LIN {X 0,Y 532.097,Z 327.827,A -85,B 0,C 180,E1 -4167.409,E2 -4167.409} C_VEL
LIN {X 0,Y 531.058,Z 327.962,A -85,B 0,C 180,E1 -4168.039,E2 -4168.039} C_VEL
LIN {X 0,Y 530.975,Z 327.968,A -85,B 0,C 180,E1 -4168.253,E2 -4168.253} C_VEL
LIN {X 0,Y 530.963,Z 327.965,A -85,B 0,C 180,E1 -4171.079,E2 -4171.079} C_VEL
LIN {X 0,Y 530.992,Z 327.968,A -85,B 0,C 180,E1 -4173.773,E2 -4173.773} C_VEL
LIN {X 0,Y 530.956,Z 327.969,A -85,B 0,C 180,E1 -4176.559,E2 -4176.559} C_VEL
LIN {X 0,Y 530.976,Z 327.967,A -85,B 0,C 180,E1 -4179.444,E2 -4179.444} C_VEL
LIN {X 0,Y 530.968,Z 327.967,A -85,B 0,C 180,E1 -4182.458,E2 -4182.458} C_VEL
LIN {X 0,Y 530.973,Z 327.971,A -85,B 0,C 180,E1 -4185.451,E2 -4185.451} C_VEL
LIN {X 0,Y 530.968,Z 327.966,A -85,B 0,C 180,E1 -4188.561,E2 -4188.561} C_VEL
LIN {X 0,Y 530.954,Z 327.976,A -85,B 0,C 180,E1 -4191.528,E2 -4191.528} C_VEL
LIN {X 0,Y 530.951,Z 327.968,A -85,B 0,C 180,E1 -4194.379,E2 -4194.379} C_VEL
LIN {X 0,Y 530.949,Z 327.974,A -85,B 0,C 180,E1 -4197.131,E2 -4197.131} C_VEL
LIN {X 0,Y 530.937,Z 327.974,A -85,B 0,C 180,E1 -4199.8,E2 -4199.8} C_VEL
LIN {X 0,Y 530.958,Z 327.969,A -85,B 0,C 180,E1 -4202.479,E2 -4202.479} C_VEL
LIN {X 0,Y 530.948,Z 327.975,A -85,B 0,C 180,E1 -4205.773,E2 -4205.773} C_VEL
LIN {X 0,Y 530.99,Z 328.027,A -85,B 0,C 180,E1 -4206.376,E2 -4206.376} C_VEL
LIN {X 0,Y 532.426,Z 335.68,A -85,B 0,C 180,E1 -4207.685,E2 -4207.685} C_VEL
LIN {X 0,Y 532.144,Z 349.705,A -85,B 0,C 180,E1 -4209.916,E2 -4209.916} C_VEL
LIN {X 0,Y 531.819,Z 362.546,A -85,B 0,C 180,E1 -4211.93,E2 -4211.93} C_VEL
LIN {X 0,Y 533.948,Z 373.777,A -85,B 0,C 180,E1 -4212.162,E2 -4212.162} C_VEL
LIN {X 0,Y 533.273,Z 498.769,A -85,B 0,C 180,E1 -4213.883,E2 -4213.883} C_VEL
LIN {X 0,Y 533.071,Z 512.331,A -85,B 0,C 180,E1 -4214.2,E2 -4214.2} C_VEL
LIN {X 0,Y 532.83,Z 526.788,A -85,B 0,C 180,E1 -4214.703,E2 -4214.703} C_VEL
LIN {X 0,Y 532.556,Z 539.12,A -85,B 0,C 180,E1 -4215.282,E2 -4215.282} C_VEL
LIN {X 0,Y 532.195,Z 550.61,A -85,B 0,C 180,E1 -4215.956,E2 -4215.956} C_VEL
LIN {X 0,Y 531.879,Z 561.401,A -85,B 0,C 180,E1 -4216.726,E2 -4216.726} C_VEL
LIN {X 0,Y 531.585,Z 571.53,A -85,B 0,C 180,E1 -4217.593,E2 -4217.593} C_VEL
LIN {X 0,Y 531.34,Z 581.016,A -85,B 0,C 180,E1 -4218.555,E2 -4218.555} C_VEL
LIN {X 0,Y 531.011,Z 591.907,A -85,B 0,C 180,E1 -4219.899,E2 -4219.899} C_VEL
LIN {X 0,Y 530.824,Z 599.5,A -85,B 0,C 180,E1 -4221.049,E2 -4221.049} C_VEL
LIN {X 0,Y 530.706,Z 604.896,A -85,B 0,C 180,E1 -4222.006,E2 -4222.006} C_VEL
LIN {X 0,Y 530.576,Z 610.311,A -85,B 0,C 180,E1 -4223.152,E2 -4223.152} C_VEL
LIN {X 0,Y 530.567,Z 614.741,A -85,B 0,C 180,E1 -4224.297,E2 -4224.297} C_VEL
LIN {X 0,Y 530.449,Z 618.285,A -85,B 0,C 180,E1 -4225.439,E2 -4225.439} C_VEL
LIN {X 0,Y 530.498,Z 620.206,A -85,B 0,C 180,E1 -4226.201,E2 -4226.201} C_VEL
LIN {X 0,Y 530.41,Z 622.929,A -85,B 0,C 180,E1 -4227.721,E2 -4227.721} C_VEL
LIN {X 0,Y 530.34,Z 624.236,A -85,B 0,C 180,E1 -4229.24,E2 -4229.24} C_VEL
LIN {X 0,Y 530.342,Z 624.496,A -85,B 0,C 180,E1 -4229.999,E2 -4229.999} C_VEL
LIN {X 0,Y 530.357,Z 623.834,A -85,B 0,C 180,E1 -4231.518,E2 -4231.518} C_VEL
LIN {X 0,Y 530.451,Z 621.843,A -85,B 0,C 180,E1 -4233.037,E2 -4233.037} C_VEL
LIN {X 0,Y 530.497,Z 620.436,A -85,B 0,C 180,E1 -4233.797,E2 -4233.797} C_VEL
LIN {X 0,Y 530.514,Z 616.296,A -85,B 0,C 180,E1 -4235.32,E2 -4235.32} C_VEL
LIN {X 0,Y 530.555,Z 613.779,A -85,B 0,C 180,E1 -4236.082,E2 -4236.082} C_VEL
LIN {X 0,Y 530.584,Z 609.106,A -85,B 0,C 180,E1 -4237.228,E2 -4237.228} C_VEL
LIN {X 0,Y 530.774,Z 602.297,A -85,B 0,C 180,E1 -4238.565,E2 -4238.565} C_VEL
LIN {X 0,Y 530.895,Z 595.198,A -85,B 0,C 180,E1 -4239.716,E2 -4239.716} C_VEL
LIN {X 0,Y 531.112,Z 588.237,A -85,B 0,C 180,E1 -4240.675,E2 -4240.675} C_VEL
LIN {X 0,Y 531.373,Z 579.159,A -85,B 0,C 180,E1 -4241.733,E2 -4241.733} C_VEL
LIN {X 0,Y 531.673,Z 569.372,A -85,B 0,C 180,E1 -4242.694,E2 -4242.694} C_VEL
LIN {X 0,Y 531.999,Z 557.577,A -85,B 0,C 180,E1 -4243.657,E2 -4243.657} C_VEL
LIN {X 0,Y 532.405,Z 544.281,A -85,B 0,C 180,E1 -4244.524,E2 -4244.524} C_VEL
LIN {X 0,Y 532.681,Z 532.145,A -85,B 0,C 180,E1 -4245.152,E2 -4245.152} C_VEL
LIN {X 0,Y 532.957,Z 519.572,A -85,B 0,C 180,E1 -4245.658,E2 -4245.658} C_VEL
LIN {X 0,Y 533.227,Z 505.576,A -85,B 0,C 180,E1 -4246.067,E2 -4246.067} C_VEL
LIN {X 0,Y 533.387,Z 488.986,A -85,B 0,C 180,E1 -4246.357,E2 -4246.357} C_VEL
LIN {X 0,Y 533.825,Z 373.018,A -85,B 0,C 180,E1 -4247.943,E2 -4247.943} C_VEL
LIN {X 0,Y 531.823,Z 362.504,A -85,B 0,C 180,E1 -4248.166,E2 -4248.166} C_VEL
LIN {X 0,Y 532.283,Z 343.943,A -85,B 0,C 180,E1 -4251.086,E2 -4251.086} C_VEL
LIN {X 0,Y 532.334,Z 335.057,A -85,B 0,C 180,E1 -4252.51,E2 -4252.51} C_VEL
LIN {X 0,Y 530.967,Z 327.972,A -85,B 0,C 180,E1 -4253.76,E2 -4253.76} C_VEL
LIN {X 0,Y 530.94,Z 327.977,A -85,B 0,C 180,E1 -4256.746,E2 -4256.746} C_VEL
LIN {X 0,Y 530.949,Z 327.974,A -85,B 0,C 180,E1 -4259.323,E2 -4259.323} C_VEL
LIN {X 0,Y 530.95,Z 327.97,A -85,B 0,C 180,E1 -4262.097,E2 -4262.097} C_VEL
LIN {X 0,Y 530.959,Z 327.976,A -85,B 0,C 180,E1 -4264.849,E2 -4264.849} C_VEL
LIN {X 0,Y 530.953,Z 327.969,A -85,B 0,C 180,E1 -4267.507,E2 -4267.507} C_VEL
LIN {X 0,Y 530.94,Z 327.972,A -85,B 0,C 180,E1 -4270.435,E2 -4270.435} C_VEL
LIN {X 0,Y 530.916,Z 327.973,A -85,B 0,C 180,E1 -4273.497,E2 -4273.497} C_VEL
LIN {X 0,Y 530.928,Z 327.974,A -85,B 0,C 180,E1 -4276.501,E2 -4276.501} C_VEL
LIN {X 0,Y 530.942,Z 327.97,A -85,B 0,C 180,E1 -4279.563,E2 -4279.563} C_VEL
LIN {X 0,Y 530.952,Z 327.97,A -85,B 0,C 180,E1 -4282.577,E2 -4282.577} C_VEL
LIN {X 0,Y 530.955,Z 327.968,A -85,B 0,C 180,E1 -4285.307,E2 -4285.307} C_VEL
LIN {X 0,Y 530.944,Z 327.965,A -85,B 0,C 180,E1 -4288.03,E2 -4288.03} C_VEL
LIN {X 0,Y 530.949,Z 327.974,A -85,B 0,C 180,E1 -4290.878,E2 -4290.878} C_VEL
LIN {X 0,Y 530.94,Z 327.965,A -85,B 0,C 180,E1 -4293.253,E2 -4293.253} C_VEL
LIN {X 0,Y 530.939,Z 327.969,A -85,B 0,C 180,E1 -4295.968,E2 -4295.968} C_VEL
LIN {X 0,Y 530.979,Z 327.964,A -85,B 0,C 180,E1 -4299.061,E2 -4299.061} C_VEL
LIN {X 0,Y 530.955,Z 327.963,A -85,B 0,C 180,E1 -4301.477,E2 -4301.477} C_VEL
LIN {X 0,Y 530.968,Z 327.974,A -85,B 0,C 180,E1 -4304.649,E2 -4304.649} C_VEL
LIN {X 0,Y 531,Z 327.961,A -85,B 0,C 180,E1 -4307.774,E2 -4307.774} C_VEL
LIN {X 0,Y 530.95,Z 327.969,A -85,B 0,C 180,E1 -4310.091,E2 -4310.091} C_VEL
LIN {X 0,Y 530.994,Z 327.967,A -85,B 0,C 180,E1 -4312.394,E2 -4312.394} C_VEL
LIN {X 0,Y 531.068,Z 327.959,A -85,B 0,C 180,E1 -4314.685,E2 -4314.685} C_VEL
LIN {X 0,Y 531.11,Z 327.948,A -85,B 0,C 180,E1 -4317.725,E2 -4317.725} C_VEL
LIN {X 0,Y 531.134,Z 327.951,A -85,B 0,C 180,E1 -4320.758,E2 -4320.758} C_VEL
LIN {X 0,Y 531.07,Z 327.954,A -85,B 0,C 180,E1 -4323.034,E2 -4323.034} C_VEL
LIN {X 0,Y 531.026,Z 327.961,A -85,B 0,C 180,E1 -4326.078,E2 -4326.078} C_VEL
LIN {X 0,Y 530.986,Z 327.964,A -85,B 0,C 180,E1 -4329.139,E2 -4329.139} C_VEL
LIN {X 0,Y 530.998,Z 327.967,A -85,B 0,C 180,E1 -4332.226,E2 -4332.226} C_VEL
LIN {X 0,Y 530.97,Z 327.965,A -85,B 0,C 180,E1 -4335.35,E2 -4335.35} C_VEL
LIN {X 0,Y 530.955,Z 327.975,A -85,B 0,C 180,E1 -4338.522,E2 -4338.522} C_VEL
LIN {X 0,Y 530.982,Z 327.962,A -85,B 0,C 180,E1 -4340.939,E2 -4340.939} C_VEL
LIN {X 0,Y 530.935,Z 327.973,A -85,B 0,C 180,E1 -4344.227,E2 -4344.227} C_VEL
LIN {X 0,Y 530.934,Z 327.972,A -85,B 0,C 180,E1 -4346.748,E2 -4346.748} C_VEL
LIN {X 0,Y 530.963,Z 327.962,A -85,B 0,C 180,E1 -4349.324,E2 -4349.324} C_VEL
LIN {X 0,Y 530.941,Z 327.974,A -85,B 0,C 180,E1 -4352.099,E2 -4352.099} C_VEL
LIN {X 0,Y 530.942,Z 327.971,A -85,B 0,C 180,E1 -4354.85,E2 -4354.85} C_VEL
LIN {X 0,Y 530.916,Z 327.973,A -85,B 0,C 180,E1 -4357.512,E2 -4357.512} C_VEL
LIN {X 0,Y 530.904,Z 327.98,A -85,B 0,C 180,E1 -4360.44,E2 -4360.44} C_VEL
LIN {X 0,Y 530.914,Z 327.973,A -85,B 0,C 180,E1 -4363.5,E2 -4363.5} C_VEL
LIN {X 0,Y 530.95,Z 327.97,A -85,B 0,C 180,E1 -4365.625,E2 -4365.625} C_VEL
LIN {X 0,Y 530.897,Z 327.98,A -85,B 0,C 180,E1 -4368.557,E2 -4368.557} C_VEL
LIN {X 0,Y 530.921,Z 327.973,A -85,B 0,C 180,E1 -4371.528,E2 -4371.528} C_VEL
LIN {X 0,Y 530.919,Z 327.979,A -85,B 0,C 180,E1 -4374.379,E2 -4374.379} C_VEL
LIN {X 0,Y 530.946,Z 327.969,A -85,B 0,C 180,E1 -4377.134,E2 -4377.134} C_VEL
LIN {X 0,Y 530.939,Z 327.974,A -85,B 0,C 180,E1 -4379.803,E2 -4379.803} C_VEL
LIN {X 0,Y 530.947,Z 327.974,A -85,B 0,C 180,E1 -4382.482,E2 -4382.482} C_VEL
LIN {X 0,Y 530.987,Z 328.019,A -85,B 0,C 180,E1 -4385.231,E2 -4385.231} C_VEL
LIN {X 0,Y 532.666,Z 336.952,A -85,B 0,C 180,E1 -4386.684,E2 -4386.684} C_VEL
LIN {X 0,Y 532.256,Z 355.336,A -85,B 0,C 180,E1 -4389.448,E2 -4389.448} C_VEL
LIN {X 0,Y 531.861,Z 371.775,A -85,B 0,C 180,E1 -4391.88,E2 -4391.88} C_VEL
LIN {X 0,Y 533.925,Z 383.626,A -85,B 0,C 180,E1 -4392.12,E2 -4392.12} C_VEL
LIN {X 0,Y 533.281,Z 508.566,A -85,B 0,C 180,E1 -4393.837,E2 -4393.837} C_VEL
LIN {X 0,Y 533.082,Z 523.14,A -85,B 0,C 180,E1 -4394.187,E2 -4394.187} C_VEL
LIN {X 0,Y 532.839,Z 536.02,A -85,B 0,C 180,E1 -4394.638,E2 -4394.638} C_VEL
LIN {X 0,Y 532.557,Z 548.002,A -85,B 0,C 180,E1 -4395.187,E2 -4395.187} C_VEL
LIN {X 0,Y 532.167,Z 561.163,A -85,B 0,C 180,E1 -4395.957,E2 -4395.957} C_VEL
LIN {X 0,Y 531.821,Z 573.057,A -85,B 0,C 180,E1 -4396.824,E2 -4396.824} C_VEL
LIN {X 0,Y 531.473,Z 583.923,A -85,B 0,C 180,E1 -4397.786,E2 -4397.786} C_VEL
LIN {X 0,Y 531.233,Z 594.661,A -85,B 0,C 180,E1 -4398.942,E2 -4398.942} C_VEL
LIN {X 0,Y 530.932,Z 603.524,A -85,B 0,C 180,E1 -4400.092,E2 -4400.092} C_VEL
LIN {X 0,Y 530.755,Z 612.018,A -85,B 0,C 180,E1 -4401.434,E2 -4401.434} C_VEL
LIN {X 0,Y 530.585,Z 618.859,A -85,B 0,C 180,E1 -4402.772,E2 -4402.772} C_VEL
LIN {X 0,Y 530.584,Z 624.963,A -85,B 0,C 180,E1 -4404.3,E2 -4404.3} C_VEL
LIN {X 0,Y 530.449,Z 628.45,A -85,B 0,C 180,E1 -4405.442,E2 -4405.442} C_VEL
LIN {X 0,Y 530.452,Z 631.838,A -85,B 0,C 180,E1 -4406.963,E2 -4406.963} C_VEL
LIN {X 0,Y 530.357,Z 633.838,A -85,B 0,C 180,E1 -4408.482,E2 -4408.482} C_VEL
LIN {X 0,Y 530.341,Z 634.5,A -85,B 0,C 180,E1 -4410.001,E2 -4410.001} C_VEL
LIN {X 0,Y 530.357,Z 633.834,A -85,B 0,C 180,E1 -4411.52,E2 -4411.52} C_VEL
LIN {X 0,Y 530.452,Z 631.83,A -85,B 0,C 180,E1 -4413.039,E2 -4413.039} C_VEL
LIN {X 0,Y 530.449,Z 628.44,A -85,B 0,C 180,E1 -4414.561,E2 -4414.561} C_VEL
LIN {X 0,Y 530.537,Z 623.565,A -85,B 0,C 180,E1 -4416.084,E2 -4416.084} C_VEL
LIN {X 0,Y 530.642,Z 617.036,A -85,B 0,C 180,E1 -4417.612,E2 -4417.612} C_VEL
LIN {X 0,Y 530.812,Z 609.768,A -85,B 0,C 180,E1 -4418.951,E2 -4418.951} C_VEL
LIN {X 0,Y 531.019,Z 600.768,A -85,B 0,C 180,E1 -4420.293,E2 -4420.293} C_VEL
LIN {X 0,Y 531.307,Z 591.32,A -85,B 0,C 180,E1 -4421.445,E2 -4421.445} C_VEL
LIN {X 0,Y 531.581,Z 580.861,A -85,B 0,C 180,E1 -4422.504,E2 -4422.504} C_VEL
LIN {X 0,Y 531.931,Z 569.317,A -85,B 0,C 180,E1 -4423.467,E2 -4423.467} C_VEL
LIN {X 0,Y 532.307,Z 556.508,A -85,B 0,C 180,E1 -4424.334,E2 -4424.334} C_VEL
LIN {X 0,Y 532.616,Z 544.007,A -85,B 0,C 180,E1 -4425.009,E2 -4425.009} C_VEL
LIN {X 0,Y 532.95,Z 530.331,A -85,B 0,C 180,E1 -4425.578,E2 -4425.578} C_VEL
LIN {X 0,Y 533.214,Z 516.18,A -85,B 0,C 180,E1 -4426.001,E2 -4426.001} C_VEL
LIN {X 0,Y 533.348,Z 502.389,A -85,B 0,C 180,E1 -4426.262,E2 -4426.262} C_VEL
LIN {X 0,Y 533.893,Z 383.182,A -85,B 0,C 180,E1 -4427.888,E2 -4427.888} C_VEL
LIN {X 0,Y 531.827,Z 371.698,A -85,B 0,C 180,E1 -4428.132,E2 -4428.132} C_VEL
LIN {X 0,Y 532.332,Z 351.756,A -85,B 0,C 180,E1 -4431.087,E2 -4431.087} C_VEL
LIN {X 0,Y 532.692,Z 336.936,A -85,B 0,C 180,E1 -4433.317,E2 -4433.317} C_VEL
LIN {X 0,Y 530.96,Z 327.973,A -85,B 0,C 180,E1 -4434.799,E2 -4434.799} C_VEL
LIN {X 0,Y 530.953,Z 327.976,A -85,B 0,C 180,E1 -4437.6,E2 -4437.6} C_VEL
LIN {X 0,Y 530.963,Z 327.968,A -85,B 0,C 180,E1 -4440.643,E2 -4440.643} C_VEL
LIN {X 0,Y 530.991,Z 327.967,A -85,B 0,C 180,E1 -4443.773,E2 -4443.773} C_VEL
LIN {X 0,Y 530.955,Z 327.969,A -85,B 0,C 180,E1 -4446.559,E2 -4446.559} C_VEL
LIN {X 0,Y 530.992,Z 327.967,A -85,B 0,C 180,E1 -4449.444,E2 -4449.444} C_VEL
LIN {X 0,Y 530.983,Z 327.967,A -85,B 0,C 180,E1 -4452.457,E2 -4452.457} C_VEL
LIN {X 0,Y 530.99,Z 327.964,A -85,B 0,C 180,E1 -4455.622,E2 -4455.622} C_VEL
LIN {X 0,Y 530.998,Z 327.969,A -85,B 0,C 180,E1 -4458.565,E2 -4458.565} C_VEL
LIN {X 0,Y 530.959,Z 327.967,A -85,B 0,C 180,E1 -4461.529,E2 -4461.529} C_VEL
LIN {X 0,Y 530.955,Z 327.976,A -85,B 0,C 180,E1 -4464.38,E2 -4464.38} C_VEL
LIN {X 0,Y 530.972,Z 327.967,A -85,B 0,C 180,E1 -4467.134,E2 -4467.134} C_VEL
LIN {X 0,Y 530.973,Z 327.971,A -85,B 0,C 180,E1 -4469.803,E2 -4469.803} C_VEL
LIN {X 0,Y 530.967,Z 327.973,A -85,B 0,C 180,E1 -4472.478,E2 -4472.478} C_VEL
LIN {X 0,Y 530.953,Z 327.97,A -85,B 0,C 180,E1 -4474.94,E2 -4474.94} C_VEL
LIN {X 0,Y 531.01,Z 328.064,A -85,B 0,C 180,E1 -4477.727,E2 -4477.727} C_VEL
LIN {X 0,Y 531.898,Z 334.003,A -85,B 0,C 180,E1 -4478.693,E2 -4478.693} C_VEL
LIN {X 0,Y 531.705,Z 352.894,A -85,B 0,C 180,E1 -4481.693,E2 -4481.693} C_VEL
LIN {X 0,Y 531.526,Z 365.213,A -85,B 0,C 180,E1 -4483.682,E2 -4483.682} C_VEL
LIN {X 0,Y 531.36,Z 373.68,A -85,B 0,C 180,E1 -4485.109,E2 -4485.109} C_VEL
LIN {X 0,Y 532.805,Z 383.09,A -85,B 0,C 180,E1 -4485.296,E2 -4485.296} C_VEL
LIN {X 0,Y 532.327,Z 480.991,A -85,B 0,C 180,E1 -4486.666,E2 -4486.666} C_VEL
LIN {X 0,Y 532.189,Z 494.465,A -85,B 0,C 180,E1 -4487.002,E2 -4487.002} C_VEL
LIN {X 0,Y 531.981,Z 506.626,A -85,B 0,C 180,E1 -4487.458,E2 -4487.458} C_VEL
LIN {X 0,Y 531.77,Z 518.851,A -85,B 0,C 180,E1 -4488.081,E2 -4488.081} C_VEL
LIN {X 0,Y 531.541,Z 530.473,A -85,B 0,C 180,E1 -4488.85,E2 -4488.85} C_VEL
LIN {X 0,Y 531.248,Z 540.771,A -85,B 0,C 180,E1 -4489.712,E2 -4489.712} C_VEL
LIN {X 0,Y 531.073,Z 550.146,A -85,B 0,C 180,E1 -4490.671,E2 -4490.671} C_VEL
LIN {X 0,Y 530.853,Z 557.738,A -85,B 0,C 180,E1 -4491.626,E2 -4491.626} C_VEL
LIN {X 0,Y 530.703,Z 565.237,A -85,B 0,C 180,E1 -4492.773,E2 -4492.773} C_VEL
LIN {X 0,Y 530.63,Z 571.198,A -85,B 0,C 180,E1 -4493.918,E2 -4493.918} C_VEL
LIN {X 0,Y 530.469,Z 575.952,A -85,B 0,C 180,E1 -4495.06,E2 -4495.06} C_VEL
LIN {X 0,Y 530.517,Z 579.514,A -85,B 0,C 180,E1 -4496.202,E2 -4496.202} C_VEL
LIN {X 0,Y 530.471,Z 581.366,A -85,B 0,C 180,E1 -4496.962,E2 -4496.962} C_VEL
LIN {X 0,Y 530.362,Z 583.823,A -85,B 0,C 180,E1 -4498.481,E2 -4498.481} C_VEL
LIN {X 0,Y 530.345,Z 584.454,A -85,B 0,C 180,E1 -4499.241,E2 -4499.241} C_VEL
LIN {X 0,Y 530.345,Z 584.674,A -85,B 0,C 180,E1 -4500,E2 -4500} C_VEL
LIN {X 0,Y 530.345,Z 584.483,A -85,B 0,C 180,E1 -4500.759,E2 -4500.759} C_VEL
LIN {X 0,Y 530.41,Z 582.917,A -85,B 0,C 180,E1 -4502.278,E2 -4502.278} C_VEL
LIN {X 0,Y 530.458,Z 581.543,A -85,B 0,C 180,E1 -4503.038,E2 -4503.038} C_VEL
LIN {X 0,Y 530.523,Z 578.711,A -85,B 0,C 180,E1 -4504.178,E2 -4504.178} C_VEL
LIN {X 0,Y 530.524,Z 574.814,A -85,B 0,C 180,E1 -4505.321,E2 -4505.321} C_VEL
LIN {X 0,Y 530.622,Z 568.966,A -85,B 0,C 180,E1 -4506.631,E2 -4506.631} C_VEL
LIN {X 0,Y 530.773,Z 562.224,A -85,B 0,C 180,E1 -4507.8,E2 -4507.8} C_VEL
LIN {X 0,Y 530.922,Z 554.043,A -85,B 0,C 180,E1 -4508.948,E2 -4508.948} C_VEL
LIN {X 0,Y 531.117,Z 545.592,A -85,B 0,C 180,E1 -4509.906,E2 -4509.906} C_VEL
LIN {X 0,Y 531.387,Z 535.209,A -85,B 0,C 180,E1 -4510.863,E2 -4510.863} C_VEL
LIN {X 0,Y 531.655,Z 524.494,A -85,B 0,C 180,E1 -4511.66,E2 -4511.66} C_VEL
LIN {X 0,Y 531.864,Z 513.565,A -85,B 0,C 180,E1 -4512.303,E2 -4512.303} C_VEL
LIN {X 0,Y 532.092,Z 500.687,A -85,B 0,C 180,E1 -4512.879,E2 -4512.879} C_VEL
LIN {X 0,Y 532.28,Z 487.641,A -85,B 0,C 180,E1 -4513.287,E2 -4513.287} C_VEL
LIN {X 0,Y 532.411,Z 473.759,A -85,B 0,C 180,E1 -4513.551,E2 -4513.551} C_VEL
LIN {X 0,Y 532.695,Z 381.43,A -85,B 0,C 180,E1 -4514.822,E2 -4514.822} C_VEL
LIN {X 0,Y 531.35,Z 373.456,A -85,B 0,C 180,E1 -4514.991,E2 -4514.991} C_VEL
LIN {X 0,Y 531.641,Z 356.128,A -85,B 0,C 180,E1 -4517.86,E2 -4517.86} C_VEL
LIN {X 0,Y 531.977,Z 337.651,A -85,B 0,C 180,E1 -4520.898,E2 -4520.898} C_VEL
LIN {X 0,Y 531.631,Z 331.341,A -85,B 0,C 180,E1 -4521.958,E2 -4521.958} C_VEL
LIN {X 0,Y 531,Z 327.97,A -85,B 0,C 180,E1 -4522.571,E2 -4522.571} C_VEL
LIN {X 0,Y 531.017,Z 327.965,A -85,B 0,C 180,E1 -4525.897,E2 -4525.897} C_VEL
LIN {X 0,Y 530.975,Z 327.968,A -85,B 0,C 180,E1 -4528.253,E2 -4528.253} C_VEL
LIN {X 0,Y 530.314,Z 328.054,A -85,B 0,C 180,E1 -4528.885,E2 -4528.885} C_VEL
LIN {X 0,Y 527.468,Z 328.408,A -85,B 0,C 180,E1 -4529.913,E2 -4529.913} C_VEL
LIN {X 0,Y 525.054,Z 328.706,A -85,B 0,C 180,E1 -4530.74,E2 -4530.74} C_VEL
LIN {X 0,Y 524.012,Z 328.833,A -85,B 0,C 180,E1 -4531.379,E2 -4531.379} C_VEL
LIN {X 0,Y 523.924,Z 328.844,A -85,B 0,C 180,E1 -4531.595,E2 -4531.595} C_VEL
LIN {X 0,Y 523.937,Z 328.847,A -85,B 0,C 180,E1 -4534.29,E2 -4534.29} C_VEL
LIN {X 0,Y 523.909,Z 328.845,A -85,B 0,C 180,E1 -4537.132,E2 -4537.132} C_VEL
LIN {X 0,Y 523.918,Z 328.849,A -85,B 0,C 180,E1 -4540.126,E2 -4540.126} C_VEL
LIN {X 0,Y 523.927,Z 328.844,A -85,B 0,C 180,E1 -4542.457,E2 -4542.457} C_VEL
LIN {X 0,Y 523.943,Z 328.845,A -85,B 0,C 180,E1 -4545.31,E2 -4545.31} C_VEL
LIN {X 0,Y 523.928,Z 328.843,A -85,B 0,C 180,E1 -4548.694,E2 -4548.694} C_VEL
LIN {X 0,Y 523.907,Z 328.85,A -85,B 0,C 180,E1 -4551.897,E2 -4551.897} C_VEL
LIN {X 0,Y 523.921,Z 328.846,A -85,B 0,C 180,E1 -4554.912,E2 -4554.912} C_VEL
LIN {X 0,Y 523.903,Z 328.852,A -85,B 0,C 180,E1 -4557.686,E2 -4557.686} C_VEL
LIN {X 0,Y 523.935,Z 328.845,A -85,B 0,C 180,E1 -4560.681,E2 -4560.681} C_VEL
LIN {X 0,Y 523.881,Z 328.854,A -85,B 0,C 180,E1 -4563.723,E2 -4563.723} C_VEL
LIN {X 0,Y 523.944,Z 328.855,A -85,B 0,C 180,E1 -4566.166,E2 -4566.166} C_VEL
LIN {X 0,Y 525.549,Z 337.744,A -85,B 0,C 180,E1 -4567.704,E2 -4567.704} C_VEL
LIN {X 0,Y 525.115,Z 353.578,A -85,B 0,C 180,E1 -4570.248,E2 -4570.248} C_VEL
LIN {X 0,Y 524.903,Z 362.629,A -85,B 0,C 180,E1 -4571.685,E2 -4571.685} C_VEL
LIN {X 0,Y 527.21,Z 375.245,A -85,B 0,C 180,E1 -4571.946,E2 -4571.946} C_VEL
LIN {X 0,Y 526.462,Z 500.288,A -85,B 0,C 180,E1 -4573.694,E2 -4573.694} C_VEL
LIN {X 0,Y 526.182,Z 514.907,A -85,B 0,C 180,E1 -4574.064,E2 -4574.064} C_VEL
LIN {X 0,Y 525.899,Z 529.12,A -85,B 0,C 180,E1 -4574.596,E2 -4574.596} C_VEL
LIN {X 0,Y 525.631,Z 540.988,A -85,B 0,C 180,E1 -4575.183,E2 -4575.183} C_VEL
LIN {X 0,Y 525.172,Z 553.604,A -85,B 0,C 180,E1 -4575.962,E2 -4575.962} C_VEL
LIN {X 0,Y 524.801,Z 566.277,A -85,B 0,C 180,E1 -4576.938,E2 -4576.938} C_VEL
LIN {X 0,Y 524.448,Z 576.751,A -85,B 0,C 180,E1 -4577.928,E2 -4577.928} C_VEL
LIN {X 0,Y 524.2,Z 586.052,A -85,B 0,C 180,E1 -4578.985,E2 -4578.985} C_VEL
LIN {X 0,Y 523.895,Z 594.661,A -85,B 0,C 180,E1 -4580.151,E2 -4580.151} C_VEL
LIN {X 0,Y 523.715,Z 601.848,A -85,B 0,C 180,E1 -4581.316,E2 -4581.316} C_VEL
LIN {X 0,Y 523.541,Z 608.743,A -85,B 0,C 180,E1 -4582.672,E2 -4582.672} C_VEL
LIN {X 0,Y 523.481,Z 614.831,A -85,B 0,C 180,E1 -4584.22,E2 -4584.22} C_VEL
LIN {X 0,Y 523.353,Z 618.372,A -85,B 0,C 180,E1 -4585.377,E2 -4585.377} C_VEL
LIN {X 0,Y 523.42,Z 620.275,A -85,B 0,C 180,E1 -4586.149,E2 -4586.149} C_VEL
LIN {X 0,Y 523.334,Z 622.991,A -85,B 0,C 180,E1 -4587.69,E2 -4587.69} C_VEL
LIN {X 0,Y 523.246,Z 624.3,A -85,B 0,C 180,E1 -4589.229,E2 -4589.229} C_VEL
LIN {X 0,Y 523.245,Z 624.544,A -85,B 0,C 180,E1 -4589.999,E2 -4589.999} C_VEL
LIN {X 0,Y 523.271,Z 623.893,A -85,B 0,C 180,E1 -4591.538,E2 -4591.538} C_VEL
LIN {X 0,Y 523.362,Z 621.913,A -85,B 0,C 180,E1 -4593.078,E2 -4593.078} C_VEL
LIN {X 0,Y 523.419,Z 620.489,A -85,B 0,C 180,E1 -4593.848,E2 -4593.848} C_VEL
LIN {X 0,Y 523.448,Z 616.381,A -85,B 0,C 180,E1 -4595.392,E2 -4595.392} C_VEL
LIN {X 0,Y 523.487,Z 612.36,A -85,B 0,C 180,E1 -4596.546,E2 -4596.546} C_VEL
LIN {X 0,Y 523.589,Z 607.34,A -85,B 0,C 180,E1 -4597.713,E2 -4597.713} C_VEL
LIN {X 0,Y 523.727,Z 601.259,A -85,B 0,C 180,E1 -4598.876,E2 -4598.876} C_VEL
LIN {X 0,Y 523.886,Z 593.962,A -85,B 0,C 180,E1 -4600.042,E2 -4600.042} C_VEL
LIN {X 0,Y 524.226,Z 585.231,A -85,B 0,C 180,E1 -4601.208,E2 -4601.208} C_VEL
LIN {X 0,Y 524.531,Z 574.611,A -85,B 0,C 180,E1 -4602.378,E2 -4602.378} C_VEL
LIN {X 0,Y 524.918,Z 562.676,A -85,B 0,C 180,E1 -4603.451,E2 -4603.451} C_VEL
LIN {X 0,Y 525.296,Z 550.638,A -85,B 0,C 180,E1 -4604.329,E2 -4604.329} C_VEL
LIN {X 0,Y 525.709,Z 537.267,A -85,B 0,C 180,E1 -4605.11,E2 -4605.11} C_VEL
LIN {X 0,Y 526.077,Z 523.353,A -85,B 0,C 180,E1 -4605.729,E2 -4605.729} C_VEL
LIN {X 0,Y 526.319,Z 509.807,A -85,B 0,C 180,E1 -4606.171,E2 -4606.171} C_VEL
LIN {X 0,Y 526.498,Z 495.634,A -85,B 0,C 180,E1 -4606.477,E2 -4606.477} C_VEL
LIN {X 0,Y 527.212,Z 374.976,A -85,B 0,C 180,E1 -4608.148,E2 -4608.148} C_VEL
LIN {X 0,Y 524.901,Z 362.492,A -85,B 0,C 180,E1 -4608.427,E2 -4608.427} C_VEL
LIN {X 0,Y 525.379,Z 343.995,A -85,B 0,C 180,E1 -4611.377,E2 -4611.377} C_VEL
LIN {X 0,Y 525.402,Z 336.262,A -85,B 0,C 180,E1 -4612.635,E2 -4612.635} C_VEL
LIN {X 0,Y 523.919,Z 328.85,A -85,B 0,C 180,E1 -4613.938,E2 -4613.938} C_VEL
LIN {X 0,Y 523.889,Z 328.856,A -85,B 0,C 180,E1 -4617.135,E2 -4617.135} C_VEL
LIN {X 0,Y 523.879,Z 328.852,A -85,B 0,C 180,E1 -4619.758,E2 -4619.758} C_VEL
LIN {X 0,Y 523.923,Z 328.848,A -85,B 0,C 180,E1 -4622.448,E2 -4622.448} C_VEL
LIN {X 0,Y 523.91,Z 328.851,A -85,B 0,C 180,E1 -4625.226,E2 -4625.226} C_VEL
LIN {X 0,Y 523.902,Z 328.846,A -85,B 0,C 180,E1 -4628.101,E2 -4628.101} C_VEL
LIN {X 0,Y 523.907,Z 328.849,A -85,B 0,C 180,E1 -4631.304,E2 -4631.304} C_VEL
LIN {X 0,Y 523.924,Z 328.849,A -85,B 0,C 180,E1 -4634.688,E2 -4634.688} C_VEL
LIN {X 0,Y 523.897,Z 328.846,A -85,B 0,C 180,E1 -4637.875,E2 -4637.875} C_VEL
LIN {X 0,Y 523.901,Z 328.848,A -85,B 0,C 180,E1 -4641.08,E2 -4641.08} C_VEL
LIN {X 0,Y 523.881,Z 328.848,A -85,B 0,C 180,E1 -4643.824,E2 -4643.824} C_VEL
LIN {X 0,Y 523.899,Z 328.852,A -85,B 0,C 180,E1 -4646.632,E2 -4646.632} C_VEL
LIN {X 0,Y 523.924,Z 328.844,A -85,B 0,C 180,E1 -4649.353,E2 -4649.353} C_VEL
LIN {X 0,Y 523.904,Z 328.847,A -85,B 0,C 180,E1 -4652.293,E2 -4652.293} C_VEL
LIN {X 0,Y 523.89,Z 328.847,A -85,B 0,C 180,E1 -4655.426,E2 -4655.426} C_VEL
LIN {X 0,Y 523.922,Z 328.843,A -85,B 0,C 180,E1 -4657.939,E2 -4657.939} C_VEL
LIN {X 0,Y 523.947,Z 328.841,A -85,B 0,C 180,E1 -4660.407,E2 -4660.407} C_VEL
LIN {X 0,Y 523.923,Z 328.849,A -85,B 0,C 180,E1 -4662.836,E2 -4662.836} C_VEL
LIN {X 0,Y 523.945,Z 328.842,A -85,B 0,C 180,E1 -4665.235,E2 -4665.235} C_VEL
LIN {X 0,Y 523.998,Z 328.838,A -85,B 0,C 180,E1 -4668.394,E2 -4668.394} C_VEL
LIN {X 0,Y 523.965,Z 328.836,A -85,B 0,C 180,E1 -4671.515,E2 -4671.515} C_VEL
LIN {X 0,Y 524.014,Z 328.838,A -85,B 0,C 180,E1 -4674.613,E2 -4674.613} C_VEL
LIN {X 0,Y 524.083,Z 328.823,A -85,B 0,C 180,E1 -4677.694,E2 -4677.694} C_VEL
LIN {X 0,Y 524.104,Z 328.826,A -85,B 0,C 180,E1 -4680.768,E2 -4680.768} C_VEL
LIN {X 0,Y 524.01,Z 328.833,A -85,B 0,C 180,E1 -4683.075,E2 -4683.075} C_VEL
LIN {X 0,Y 523.988,Z 328.838,A -85,B 0,C 180,E1 -4686.16,E2 -4686.16} C_VEL
LIN {X 0,Y 523.935,Z 328.841,A -85,B 0,C 180,E1 -4689.263,E2 -4689.263} C_VEL
LIN {X 0,Y 523.937,Z 328.849,A -85,B 0,C 180,E1 -4692.393,E2 -4692.393} C_VEL
LIN {X 0,Y 523.908,Z 328.845,A -85,B 0,C 180,E1 -4695.563,E2 -4695.563} C_VEL
LIN {X 0,Y 523.9,Z 328.847,A -85,B 0,C 180,E1 -4697.971,E2 -4697.971} C_VEL
LIN {X 0,Y 523.957,Z 328.844,A -85,B 0,C 180,E1 -4700.411,E2 -4700.411} C_VEL
LIN {X 0,Y 523.892,Z 328.846,A -85,B 0,C 180,E1 -4702.894,E2 -4702.894} C_VEL
LIN {X 0,Y 523.881,Z 328.848,A -85,B 0,C 180,E1 -4705.422,E2 -4705.422} C_VEL
LIN {X 0,Y 523.897,Z 328.849,A -85,B 0,C 180,E1 -4708.003,E2 -4708.003} C_VEL
LIN {X 0,Y 523.901,Z 328.85,A -85,B 0,C 180,E1 -4710.648,E2 -4710.648} C_VEL
LIN {X 0,Y 523.912,Z 328.845,A -85,B 0,C 180,E1 -4713.73,E2 -4713.73} C_VEL
LIN {X 0,Y 523.847,Z 328.861,A -85,B 0,C 180,E1 -4716.396,E2 -4716.396} C_VEL
LIN {X 0,Y 523.891,Z 328.848,A -85,B 0,C 180,E1 -4719.087,E2 -4719.087} C_VEL
LIN {X 0,Y 523.864,Z 328.857,A -85,B 0,C 180,E1 -4722.453,E2 -4722.453} C_VEL
LIN {X 0,Y 523.919,Z 328.844,A -85,B 0,C 180,E1 -4725.313,E2 -4725.313} C_VEL
LIN {X 0,Y 523.866,Z 328.854,A -85,B 0,C 180,E1 -4728.701,E2 -4728.701} C_VEL
LIN {X 0,Y 523.879,Z 328.854,A -85,B 0,C 180,E1 -4731.897,E2 -4731.897} C_VEL
LIN {X 0,Y 523.904,Z 328.847,A -85,B 0,C 180,E1 -4734.914,E2 -4734.914} C_VEL
LIN {X 0,Y 523.893,Z 328.851,A -85,B 0,C 180,E1 -4737.687,E2 -4737.687} C_VEL
LIN {X 0,Y 523.928,Z 328.844,A -85,B 0,C 180,E1 -4740.682,E2 -4740.682} C_VEL
LIN {X 0,Y 523.876,Z 328.855,A -85,B 0,C 180,E1 -4743.725,E2 -4743.725} C_VEL
LIN {X 0,Y 523.93,Z 328.968,A -85,B 0,C 180,E1 -4745.033,E2 -4745.033} C_VEL
LIN {X 0,Y 525.768,Z 338.244,A -85,B 0,C 180,E1 -4746.569,E2 -4746.569} C_VEL
LIN {X 0,Y 525.335,Z 355.89,A -85,B 0,C 180,E1 -4749.259,E2 -4749.259} C_VEL
LIN {X 0,Y 524.918,Z 371.725,A -85,B 0,C 180,E1 -4751.635,E2 -4751.635} C_VEL
LIN {X 0,Y 527.174,Z 384.814,A -85,B 0,C 180,E1 -4751.9,E2 -4751.9} C_VEL
LIN {X 0,Y 526.459,Z 509.734,A -85,B 0,C 180,E1 -4753.646,E2 -4753.646} C_VEL
LIN {X 0,Y 526.25,Z 523.912,A -85,B 0,C 180,E1 -4754.003,E2 -4754.003} C_VEL
LIN {X 0,Y 525.962,Z 536.173,A -85,B 0,C 180,E1 -4754.442,E2 -4754.442} C_VEL
LIN {X 0,Y 525.624,Z 549.71,A -85,B 0,C 180,E1 -4755.086,E2 -4755.086} C_VEL
LIN {X 0,Y 525.21,Z 562.523,A -85,B 0,C 180,E1 -4755.866,E2 -4755.866} C_VEL
LIN {X 0,Y 524.828,Z 574.164,A -85,B 0,C 180,E1 -4756.744,E2 -4756.744} C_VEL
LIN {X 0,Y 524.444,Z 585.359,A -85,B 0,C 180,E1 -4757.771,E2 -4757.771} C_VEL
LIN {X 0,Y 524.239,Z 594.593,A -85,B 0,C 180,E1 -4758.792,E2 -4758.792} C_VEL
LIN {X 0,Y 523.887,Z 603.456,A -85,B 0,C 180,E1 -4759.958,E2 -4759.958} C_VEL
LIN {X 0,Y 523.679,Z 611.95,A -85,B 0,C 180,E1 -4761.318,E2 -4761.318} C_VEL
LIN {X 0,Y 523.503,Z 618.791,A -85,B 0,C 180,E1 -4762.674,E2 -4762.674} C_VEL
LIN {X 0,Y 523.472,Z 623.507,A -85,B 0,C 180,E1 -4763.835,E2 -4763.835} C_VEL
LIN {X 0,Y 523.376,Z 627.329,A -85,B 0,C 180,E1 -4764.994,E2 -4764.994} C_VEL
LIN {X 0,Y 523.418,Z 630.275,A -85,B 0,C 180,E1 -4766.152,E2 -4766.152} C_VEL
LIN {X 0,Y 523.333,Z 632.966,A -85,B 0,C 180,E1 -4767.692,E2 -4767.692} C_VEL
LIN {X 0,Y 523.247,Z 634.296,A -85,B 0,C 180,E1 -4769.232,E2 -4769.232} C_VEL
LIN {X 0,Y 523.247,Z 634.295,A -85,B 0,C 180,E1 -4770.771,E2 -4770.771} C_VEL
LIN {X 0,Y 523.333,Z 632.959,A -85,B 0,C 180,E1 -4772.31,E2 -4772.31} C_VEL
LIN {X 0,Y 523.419,Z 630.265,A -85,B 0,C 180,E1 -4773.851,E2 -4773.851} C_VEL
LIN {X 0,Y 523.451,Z 626.139,A -85,B 0,C 180,E1 -4775.394,E2 -4775.394} C_VEL
LIN {X 0,Y 523.496,Z 620.451,A -85,B 0,C 180,E1 -4776.941,E2 -4776.941} C_VEL
LIN {X 0,Y 523.636,Z 614.034,A -85,B 0,C 180,E1 -4778.297,E2 -4778.297} C_VEL
LIN {X 0,Y 523.863,Z 606.064,A -85,B 0,C 180,E1 -4779.655,E2 -4779.655} C_VEL
LIN {X 0,Y 524.107,Z 597.725,A -85,B 0,C 180,E1 -4780.822,E2 -4780.822} C_VEL
LIN {X 0,Y 524.45,Z 586.943,A -85,B 0,C 180,E1 -4782.069,E2 -4782.069} C_VEL
LIN {X 0,Y 524.753,Z 576.485,A -85,B 0,C 180,E1 -4783.063,E2 -4783.063} C_VEL
LIN {X 0,Y 525.195,Z 563.913,A -85,B 0,C 180,E1 -4784.038,E2 -4784.038} C_VEL
LIN {X 0,Y 525.579,Z 551.436,A -85,B 0,C 180,E1 -4784.818,E2 -4784.818} C_VEL
LIN {X 0,Y 525.933,Z 538.617,A -85,B 0,C 180,E1 -4785.453,E2 -4785.453} C_VEL
LIN {X 0,Y 526.186,Z 524.835,A -85,B 0,C 180,E1 -4785.969,E2 -4785.969} C_VEL
LIN {X 0,Y 526.476,Z 510.769,A -85,B 0,C 180,E1 -4786.331,E2 -4786.331} C_VEL
LIN {X 0,Y 526.66,Z 482.647,A -85,B 0,C 180,E1 -4786.749,E2 -4786.749} C_VEL
LIN {X 0,Y 527.074,Z 383.404,A -85,B 0,C 180,E1 -4788.123,E2 -4788.123} C_VEL
LIN {X 0,Y 524.88,Z 371.609,A -85,B 0,C 180,E1 -4788.384,E2 -4788.384} C_VEL
LIN {X 0,Y 525.439,Z 351.694,A -85,B 0,C 180,E1 -4791.377,E2 -4791.377} C_VEL
LIN {X 0,Y 525.774,Z 338.227,A -85,B 0,C 180,E1 -4793.433,E2 -4793.433} C_VEL
LIN {X 0,Y 523.915,Z 328.851,A -85,B 0,C 180,E1 -4794.997,E2 -4794.997} C_VEL
LIN {X 0,Y 523.899,Z 328.852,A -85,B 0,C 180,E1 -4798.004,E2 -4798.004} C_VEL
LIN {X 0,Y 523.938,Z 328.845,A -85,B 0,C 180,E1 -4800.853,E2 -4800.853} C_VEL
LIN {X 0,Y 523.963,Z 328.843,A -85,B 0,C 180,E1 -4803.735,E2 -4803.735} C_VEL
LIN {X 0,Y 523.903,Z 328.847,A -85,B 0,C 180,E1 -4806.401,E2 -4806.401} C_VEL
LIN {X 0,Y 523.926,Z 328.85,A -85,B 0,C 180,E1 -4809.085,E2 -4809.085} C_VEL
LIN {X 0,Y 523.956,Z 328.84,A -85,B 0,C 180,E1 -4812.119,E2 -4812.119} C_VEL
LIN {X 0,Y 523.958,Z 328.842,A -85,B 0,C 180,E1 -4815.309,E2 -4815.309} C_VEL
LIN {X 0,Y 523.961,Z 328.846,A -85,B 0,C 180,E1 -4818.69,E2 -4818.69} C_VEL
LIN {X 0,Y 523.92,Z 328.846,A -85,B 0,C 180,E1 -4821.081,E2 -4821.081} C_VEL
LIN {X 0,Y 523.9,Z 328.848,A -85,B 0,C 180,E1 -4823.825,E2 -4823.825} C_VEL
LIN {X 0,Y 523.946,Z 328.846,A -85,B 0,C 180,E1 -4826.636,E2 -4826.636} C_VEL
LIN {X 0,Y 523.96,Z 328.842,A -85,B 0,C 180,E1 -4829.356,E2 -4829.356} C_VEL
LIN {X 0,Y 523.943,Z 328.85,A -85,B 0,C 180,E1 -4832.29,E2 -4832.29} C_VEL
LIN {X 0,Y 523.906,Z 328.851,A -85,B 0,C 180,E1 -4835.427,E2 -4835.427} C_VEL
LIN {X 0,Y 523.969,Z 328.926,A -85,B 0,C 180,E1 -4837.602,E2 -4837.602} C_VEL
LIN {X 0,Y 524.939,Z 335.046,A -85,B 0,C 180,E1 -4838.603,E2 -4838.603} C_VEL
LIN {X 0,Y 524.726,Z 353.072,A -85,B 0,C 180,E1 -4841.472,E2 -4841.472} C_VEL
LIN {X 0,Y 524.545,Z 366.585,A -85,B 0,C 180,E1 -4843.658,E2 -4843.658} C_VEL
LIN {X 0,Y 524.414,Z 374.134,A -85,B 0,C 180,E1 -4844.917,E2 -4844.917} C_VEL
LIN {X 0,Y 525.938,Z 383.216,A -85,B 0,C 180,E1 -4845.1,E2 -4845.1} C_VEL
LIN {X 0,Y 525.387,Z 482.607,A -85,B 0,C 180,E1 -4846.536,E2 -4846.536} C_VEL
LIN {X 0,Y 525.241,Z 494.834,A -85,B 0,C 180,E1 -4846.852,E2 -4846.852} C_VEL
LIN {X 0,Y 525.026,Z 507.5,A -85,B 0,C 180,E1 -4847.338,E2 -4847.338} C_VEL
LIN {X 0,Y 524.784,Z 519.803,A -85,B 0,C 180,E1 -4847.98,E2 -4847.98} C_VEL
LIN {X 0,Y 524.541,Z 531.774,A -85,B 0,C 180,E1 -4848.798,E2 -4848.798} C_VEL
LIN {X 0,Y 524.22,Z 541.925,A -85,B 0,C 180,E1 -4849.67,E2 -4849.67} C_VEL
LIN {X 0,Y 524.048,Z 550.305,A -85,B 0,C 180,E1 -4850.544,E2 -4850.544} C_VEL
LIN {X 0,Y 523.829,Z 557.958,A -85,B 0,C 180,E1 -4851.513,E2 -4851.513} C_VEL
LIN {X 0,Y 523.653,Z 565.482,A -85,B 0,C 180,E1 -4852.675,E2 -4852.675} C_VEL
LIN {X 0,Y 523.564,Z 571.478,A -85,B 0,C 180,E1 -4853.835,E2 -4853.835} C_VEL
LIN {X 0,Y 523.393,Z 576.24,A -85,B 0,C 180,E1 -4854.993,E2 -4854.993} C_VEL
LIN {X 0,Y 523.444,Z 579.827,A -85,B 0,C 180,E1 -4856.151,E2 -4856.151} C_VEL
LIN {X 0,Y 523.41,Z 581.692,A -85,B 0,C 180,E1 -4856.921,E2 -4856.921} C_VEL
LIN {X 0,Y 523.335,Z 583.121,A -85,B 0,C 180,E1 -4857.691,E2 -4857.691} C_VEL
LIN {X 0,Y 523.275,Z 584.15,A -85,B 0,C 180,E1 -4858.461,E2 -4858.461} C_VEL
LIN {X 0,Y 523.253,Z 584.776,A -85,B 0,C 180,E1 -4859.23,E2 -4859.23} C_VEL
LIN {X 0,Y 523.253,Z 584.997,A -85,B 0,C 180,E1 -4860,E2 -4860} C_VEL
LIN {X 0,Y 523.253,Z 584.812,A -85,B 0,C 180,E1 -4860.77,E2 -4860.77} C_VEL
LIN {X 0,Y 523.275,Z 584.223,A -85,B 0,C 180,E1 -4861.539,E2 -4861.539} C_VEL
LIN {X 0,Y 523.398,Z 581.849,A -85,B 0,C 180,E1 -4863.079,E2 -4863.079} C_VEL
LIN {X 0,Y 523.443,Z 578.996,A -85,B 0,C 180,E1 -4864.235,E2 -4864.235} C_VEL
LIN {X 0,Y 523.463,Z 575.076,A -85,B 0,C 180,E1 -4865.393,E2 -4865.393} C_VEL
LIN {X 0,Y 523.571,Z 569.657,A -85,B 0,C 180,E1 -4866.628,E2 -4866.628} C_VEL
LIN {X 0,Y 523.725,Z 562.425,A -85,B 0,C 180,E1 -4867.906,E2 -4867.906} C_VEL
LIN {X 0,Y 523.901,Z 554.19,A -85,B 0,C 180,E1 -4869.069,E2 -4869.069} C_VEL
LIN {X 0,Y 524.105,Z 545.718,A -85,B 0,C 180,E1 -4870.039,E2 -4870.039} C_VEL
LIN {X 0,Y 524.409,Z 535.27,A -85,B 0,C 180,E1 -4871.01,E2 -4871.01} C_VEL
LIN {X 0,Y 524.686,Z 524.931,A -85,B 0,C 180,E1 -4871.787,E2 -4871.787} C_VEL
LIN {X 0,Y 524.907,Z 513.442,A -85,B 0,C 180,E1 -4872.468,E2 -4872.468} C_VEL
LIN {X 0,Y 525.133,Z 501.708,A -85,B 0,C 180,E1 -4873.003,E2 -4873.003} C_VEL
LIN {X 0,Y 525.325,Z 489.075,A -85,B 0,C 180,E1 -4873.417,E2 -4873.417} C_VEL
LIN {X 0,Y 525.481,Z 476.067,A -85,B 0,C 180,E1 -4873.684,E2 -4873.684} C_VEL
LIN {X 0,Y 525.836,Z 382.364,A -85,B 0,C 180,E1 -4875.006,E2 -4875.006} C_VEL
LIN {X 0,Y 524.366,Z 373.657,A -85,B 0,C 180,E1 -4875.201,E2 -4875.201} C_VEL
LIN {X 0,Y 524.68,Z 356.766,A -85,B 0,C 180,E1 -4878.003,E2 -4878.003} C_VEL
LIN {X 0,Y 525.005,Z 338.886,A -85,B 0,C 180,E1 -4880.963,E2 -4880.963} C_VEL
LIN {X 0,Y 524.67,Z 332.584,A -85,B 0,C 180,E1 -4882.028,E2 -4882.028} C_VEL
LIN {X 0,Y 523.957,Z 328.847,A -85,B 0,C 180,E1 -4882.69,E2 -4882.69} C_VEL
LIN {X 0,Y 523.988,Z 328.842,A -85,B 0,C 180,E1 -4886.019,E2 -4886.019} C_VEL
LIN {X 0,Y 523.934,Z 328.843,A -85,B 0,C 180,E1 -4888.875,E2 -4888.875} C_VEL
LIN {X 0,Y 523.924,Z 328.844,A -85,B 0,C 180,E1 -4891.595,E2 -4891.595} C_VEL
LIN {X 0,Y 523.253,Z 328.933,A -85,B 0,C 180,E1 -4892.237,E2 -4892.237} C_VEL
LIN {X 0,Y 520.413,Z 329.282,A -85,B 0,C 180,E1 -4893.279,E2 -4893.279} C_VEL
LIN {X 0,Y 518.01,Z 329.588,A -85,B 0,C 180,E1 -4894.118,E2 -4894.118} C_VEL
LIN {X 0,Y 516.967,Z 329.711,A -85,B 0,C 180,E1 -4894.766,E2 -4894.766} C_VEL
LIN {X 0,Y 516.877,Z 329.721,A -85,B 0,C 180,E1 -4894.986,E2 -4894.986} C_VEL
LIN {X 0,Y 516.883,Z 329.728,A -85,B 0,C 180,E1 -4897.942,E2 -4897.942} C_VEL
LIN {X 0,Y 516.869,Z 329.722,A -85,B 0,C 180,E1 -4900.743,E2 -4900.743} C_VEL
LIN {X 0,Y 516.864,Z 329.723,A -85,B 0,C 180,E1 -4902.834,E2 -4902.834} C_VEL
LIN {X 0,Y 516.901,Z 329.719,A -85,B 0,C 180,E1 -4905.007,E2 -4905.007} C_VEL
LIN {X 0,Y 516.892,Z 329.72,A -85,B 0,C 180,E1 -4908.402,E2 -4908.402} C_VEL
LIN {X 0,Y 516.878,Z 329.727,A -85,B 0,C 180,E1 -4911.283,E2 -4911.283} C_VEL
LIN {X 0,Y 516.863,Z 329.724,A -85,B 0,C 180,E1 -4914.671,E2 -4914.671} C_VEL
LIN {X 0,Y 516.868,Z 329.729,A -85,B 0,C 180,E1 -4917.462,E2 -4917.462} C_VEL
LIN {X 0,Y 516.902,Z 329.722,A -85,B 0,C 180,E1 -4920.693,E2 -4920.693} C_VEL
LIN {X 0,Y 516.858,Z 329.729,A -85,B 0,C 180,E1 -4923.824,E2 -4923.824} C_VEL
LIN {X 0,Y 516.901,Z 329.867,A -85,B 0,C 180,E1 -4925.98,E2 -4925.98} C_VEL
LIN {X 0,Y 518.475,Z 337.7,A -85,B 0,C 180,E1 -4927.365,E2 -4927.365} C_VEL
LIN {X 0,Y 518.496,Z 346.027,A -85,B 0,C 180,E1 -4928.74,E2 -4928.74} C_VEL
LIN {X 0,Y 517.955,Z 362.666,A -85,B 0,C 180,E1 -4931.425,E2 -4931.425} C_VEL
LIN {X 0,Y 520.442,Z 376.303,A -85,B 0,C 180,E1 -4931.716,E2 -4931.716} C_VEL
LIN {X 0,Y 519.665,Z 499.169,A -85,B 0,C 180,E1 -4933.449,E2 -4933.449} C_VEL
LIN {X 0,Y 519.417,Z 513.612,A -85,B 0,C 180,E1 -4933.806,E2 -4933.806} C_VEL
LIN {X 0,Y 519.165,Z 526.942,A -85,B 0,C 180,E1 -4934.291,E2 -4934.291} C_VEL
LIN {X 0,Y 518.809,Z 539.323,A -85,B 0,C 180,E1 -4934.883,E2 -4934.883} C_VEL
LIN {X 0,Y 518.35,Z 552.262,A -85,B 0,C 180,E1 -4935.673,E2 -4935.673} C_VEL
LIN {X 0,Y 517.963,Z 563.997,A -85,B 0,C 180,E1 -4936.563,E2 -4936.563} C_VEL
LIN {X 0,Y 517.519,Z 575.457,A -85,B 0,C 180,E1 -4937.623,E2 -4937.623} C_VEL
LIN {X 0,Y 517.193,Z 586.155,A -85,B 0,C 180,E1 -4938.834,E2 -4938.834} C_VEL
LIN {X 0,Y 516.874,Z 594.761,A -85,B 0,C 180,E1 -4940.016,E2 -4940.016} C_VEL
LIN {X 0,Y 516.649,Z 603.04,A -85,B 0,C 180,E1 -4941.393,E2 -4941.393} C_VEL
LIN {X 0,Y 516.475,Z 608.809,A -85,B 0,C 180,E1 -4942.571,E2 -4942.571} C_VEL
LIN {X 0,Y 516.398,Z 614.921,A -85,B 0,C 180,E1 -4944.14,E2 -4944.14} C_VEL
LIN {X 0,Y 516.264,Z 618.46,A -85,B 0,C 180,E1 -4945.314,E2 -4945.314} C_VEL
LIN {X 0,Y 516.343,Z 620.34,A -85,B 0,C 180,E1 -4946.097,E2 -4946.097} C_VEL
LIN {X 0,Y 516.26,Z 623.067,A -85,B 0,C 180,E1 -4947.658,E2 -4947.658} C_VEL
LIN {X 0,Y 516.156,Z 624.392,A -85,B 0,C 180,E1 -4949.219,E2 -4949.219} C_VEL
LIN {X 0,Y 516.153,Z 624.611,A -85,B 0,C 180,E1 -4949.999,E2 -4949.999} C_VEL
LIN {X 0,Y 516.188,Z 623.974,A -85,B 0,C 180,E1 -4951.559,E2 -4951.559} C_VEL
LIN {X 0,Y 516.276,Z 622.003,A -85,B 0,C 180,E1 -4953.12,E2 -4953.12} C_VEL
LIN {X 0,Y 516.343,Z 620.552,A -85,B 0,C 180,E1 -4953.901,E2 -4953.901} C_VEL
LIN {X 0,Y 516.381,Z 616.462,A -85,B 0,C 180,E1 -4955.466,E2 -4955.466} C_VEL
LIN {X 0,Y 516.41,Z 611.87,A -85,B 0,C 180,E1 -4956.782,E2 -4956.782} C_VEL
LIN {X 0,Y 516.575,Z 605.536,A -85,B 0,C 180,E1 -4958.212,E2 -4958.212} C_VEL
LIN {X 0,Y 516.816,Z 597.879,A -85,B 0,C 180,E1 -4959.588,E2 -4959.588} C_VEL
LIN {X 0,Y 517.094,Z 588.397,A -85,B 0,C 180,E1 -4960.968,E2 -4960.968} C_VEL
LIN {X 0,Y 517.447,Z 578.375,A -85,B 0,C 180,E1 -4962.16,E2 -4962.16} C_VEL
LIN {X 0,Y 517.824,Z 567.395,A -85,B 0,C 180,E1 -4963.239,E2 -4963.239} C_VEL
LIN {X 0,Y 518.206,Z 556.392,A -85,B 0,C 180,E1 -4964.128,E2 -4964.128} C_VEL
LIN {X 0,Y 518.642,Z 544.451,A -85,B 0,C 180,E1 -4964.918,E2 -4964.918} C_VEL
LIN {X 0,Y 519.042,Z 531.26,A -85,B 0,C 180,E1 -4965.61,E2 -4965.61} C_VEL
LIN {X 0,Y 519.374,Z 517.354,A -85,B 0,C 180,E1 -4966.161,E2 -4966.161} C_VEL
LIN {X 0,Y 519.61,Z 503.397,A -85,B 0,C 180,E1 -4966.55,E2 -4966.55} C_VEL
LIN {X 0,Y 519.788,Z 485.452,A -85,B 0,C 180,E1 -4966.848,E2 -4966.848} C_VEL
LIN {X 0,Y 520.466,Z 376.16,A -85,B 0,C 180,E1 -4968.375,E2 -4968.375} C_VEL
LIN {X 0,Y 517.95,Z 362.588,A -85,B 0,C 180,E1 -4968.678,E2 -4968.678} C_VEL
LIN {X 0,Y 518.542,Z 344.048,A -85,B 0,C 180,E1 -4971.673,E2 -4971.673} C_VEL
LIN {X 0,Y 518.406,Z 337.276,A -85,B 0,C 180,E1 -4972.798,E2 -4972.798} C_VEL
LIN {X 0,Y 516.904,Z 329.725,A -85,B 0,C 180,E1 -4974.17,E2 -4974.17} C_VEL
LIN {X 0,Y 516.832,Z 329.734,A -85,B 0,C 180,E1 -4976.661,E2 -4976.661} C_VEL
LIN {X 0,Y 516.874,Z 329.726,A -85,B 0,C 180,E1 -4979.516,E2 -4979.516} C_VEL
LIN {X 0,Y 516.885,Z 329.726,A -85,B 0,C 180,E1 -4982.541,E2 -4982.541} C_VEL
LIN {X 0,Y 516.856,Z 329.728,A -85,B 0,C 180,E1 -4985.328,E2 -4985.328} C_VEL
LIN {X 0,Y 516.867,Z 329.723,A -85,B 0,C 180,E1 -4987.941,E2 -4987.941} C_VEL
LIN {X 0,Y 516.842,Z 329.732,A -85,B 0,C 180,E1 -4990.744,E2 -4990.744} C_VEL
LIN {X 0,Y 516.87,Z 329.722,A -85,B 0,C 180,E1 -4993.902,E2 -4993.902} C_VEL
LIN {X 0,Y 516.87,Z 329.722,A -85,B 0,C 180,E1 -4996.106,E2 -4996.106} C_VEL
LIN {X 0,Y 516.843,Z 329.729,A -85,B 0,C 180,E1 -4999.254,E2 -4999.254} C_VEL
LIN {X 0,Y 516.864,Z 329.719,A -85,B 0,C 180,E1 -5002.057,E2 -5002.057} C_VEL
LIN {X 0,Y 516.86,Z 329.726,A -85,B 0,C 180,E1 -5005.173,E2 -5005.173} C_VEL
LIN {X 0,Y 516.854,Z 329.72,A -85,B 0,C 180,E1 -5007.974,E2 -5007.974} C_VEL
LIN {X 0,Y 516.889,Z 329.727,A -85,B 0,C 180,E1 -5010.693,E2 -5010.693} C_VEL
LIN {X 0,Y 516.867,Z 329.715,A -85,B 0,C 180,E1 -5013.817,E2 -5013.817} C_VEL
LIN {X 0,Y 516.841,Z 329.734,A -85,B 0,C 180,E1 -5016.775,E2 -5016.775} C_VEL
LIN {X 0,Y 516.915,Z 329.711,A -85,B 0,C 180,E1 -5019.734,E2 -5019.734} C_VEL
LIN {X 0,Y 516.878,Z 329.723,A -85,B 0,C 180,E1 -5022.594,E2 -5022.594} C_VEL
LIN {X 0,Y 516.914,Z 329.719,A -85,B 0,C 180,E1 -5025.029,E2 -5025.029} C_VEL
LIN {X 0,Y 516.951,Z 329.714,A -85,B 0,C 180,E1 -5028.233,E2 -5028.233} C_VEL
LIN {X 0,Y 516.933,Z 329.713,A -85,B 0,C 180,E1 -5031.399,E2 -5031.399} C_VEL
LIN {X 0,Y 516.964,Z 329.717,A -85,B 0,C 180,E1 -5034.539,E2 -5034.539} C_VEL
LIN {X 0,Y 517.055,Z 329.699,A -85,B 0,C 180,E1 -5037.663,E2 -5037.663} C_VEL
LIN {X 0,Y 517.074,Z 329.702,A -85,B 0,C 180,E1 -5040.779,E2 -5040.779} C_VEL
LIN {X 0,Y 516.951,Z 329.712,A -85,B 0,C 180,E1 -5043.117,E2 -5043.117} C_VEL
LIN {X 0,Y 516.954,Z 329.716,A -85,B 0,C 180,E1 -5046.244,E2 -5046.244} C_VEL
LIN {X 0,Y 516.895,Z 329.718,A -85,B 0,C 180,E1 -5049.39,E2 -5049.39} C_VEL
LIN {X 0,Y 516.889,Z 329.725,A -85,B 0,C 180,E1 -5052.565,E2 -5052.565} C_VEL
LIN {X 0,Y 516.929,Z 329.715,A -85,B 0,C 180,E1 -5055.147,E2 -5055.147} C_VEL
LIN {X 0,Y 516.862,Z 329.727,A -85,B 0,C 180,E1 -5058.224,E2 -5058.224} C_VEL
LIN {X 0,Y 516.897,Z 329.719,A -85,B 0,C 180,E1 -5060.702,E2 -5060.702} C_VEL
LIN {X 0,Y 516.869,Z 329.722,A -85,B 0,C 180,E1 -5064.074,E2 -5064.074} C_VEL
LIN {X 0,Y 516.821,Z 329.731,A -85,B 0,C 180,E1 -5066.664,E2 -5066.664} C_VEL
LIN {X 0,Y 516.883,Z 329.716,A -85,B 0,C 180,E1 -5069.522,E2 -5069.522} C_VEL
LIN {X 0,Y 516.878,Z 329.725,A -85,B 0,C 180,E1 -5072.543,E2 -5072.543} C_VEL
LIN {X 0,Y 516.836,Z 329.726,A -85,B 0,C 180,E1 -5075.328,E2 -5075.328} C_VEL
LIN {X 0,Y 516.856,Z 329.727,A -85,B 0,C 180,E1 -5078.718,E2 -5078.718} C_VEL
LIN {X 0,Y 516.822,Z 329.73,A -85,B 0,C 180,E1 -5081.784,E2 -5081.784} C_VEL
LIN {X 0,Y 516.885,Z 329.721,A -85,B 0,C 180,E1 -5085.008,E2 -5085.008} C_VEL
LIN {X 0,Y 516.819,Z 329.736,A -85,B 0,C 180,E1 -5088.411,E2 -5088.411} C_VEL
LIN {X 0,Y 516.849,Z 329.725,A -85,B 0,C 180,E1 -5091.283,E2 -5091.283} C_VEL
LIN {X 0,Y 516.841,Z 329.729,A -85,B 0,C 180,E1 -5094.675,E2 -5094.675} C_VEL
LIN {X 0,Y 516.859,Z 329.725,A -85,B 0,C 180,E1 -5097.463,E2 -5097.463} C_VEL
LIN {X 0,Y 516.878,Z 329.723,A -85,B 0,C 180,E1 -5100.483,E2 -5100.483} C_VEL
LIN {X 0,Y 516.822,Z 329.731,A -85,B 0,C 180,E1 -5103.338,E2 -5103.338} C_VEL
LIN {X 0,Y 516.853,Z 329.752,A -85,B 0,C 180,E1 -5104.802,E2 -5104.802} C_VEL
LIN {X 0,Y 518.872,Z 339.534,A -85,B 0,C 180,E1 -5106.45,E2 -5106.45} C_VEL
LIN {X 0,Y 518.467,Z 354.343,A -85,B 0,C 180,E1 -5108.741,E2 -5108.741} C_VEL
LIN {X 0,Y 517.961,Z 371.654,A -85,B 0,C 180,E1 -5111.379,E2 -5111.379} C_VEL
LIN {X 0,Y 520.437,Z 385.474,A -85,B 0,C 180,E1 -5111.668,E2 -5111.668} C_VEL
LIN {X 0,Y 519.647,Z 509.667,A -85,B 0,C 180,E1 -5113.426,E2 -5113.426} C_VEL
LIN {X 0,Y 519.406,Z 523.812,A -85,B 0,C 180,E1 -5113.786,E2 -5113.786} C_VEL
LIN {X 0,Y 519.075,Z 537.462,A -85,B 0,C 180,E1 -5114.29,E2 -5114.29} C_VEL
LIN {X 0,Y 518.709,Z 551.411,A -85,B 0,C 180,E1 -5114.983,E2 -5114.983} C_VEL
LIN {X 0,Y 518.268,Z 563.882,A -85,B 0,C 180,E1 -5115.773,E2 -5115.773} C_VEL
LIN {X 0,Y 517.806,Z 576.444,A -85,B 0,C 180,E1 -5116.761,E2 -5116.761} C_VEL
LIN {X 0,Y 517.451,Z 587.436,A -85,B 0,C 180,E1 -5117.826,E2 -5117.826} C_VEL
LIN {X 0,Y 517.1,Z 597.675,A -85,B 0,C 180,E1 -5119.032,E2 -5119.032} C_VEL
LIN {X 0,Y 516.809,Z 606.011,A -85,B 0,C 180,E1 -5120.214,E2 -5120.214} C_VEL
LIN {X 0,Y 516.581,Z 613.979,A -85,B 0,C 180,E1 -5121.592,E2 -5121.592} C_VEL
LIN {X 0,Y 516.401,Z 620.391,A -85,B 0,C 180,E1 -5122.966,E2 -5122.966} C_VEL
LIN {X 0,Y 516.407,Z 624.834,A -85,B 0,C 180,E1 -5124.143,E2 -5124.143} C_VEL
LIN {X 0,Y 516.264,Z 628.329,A -85,B 0,C 180,E1 -5125.316,E2 -5125.316} C_VEL
LIN {X 0,Y 516.324,Z 630.207,A -85,B 0,C 180,E1 -5126.099,E2 -5126.099} C_VEL
LIN {X 0,Y 516.259,Z 632.899,A -85,B 0,C 180,E1 -5127.661,E2 -5127.661} C_VEL
LIN {X 0,Y 516.157,Z 634.229,A -85,B 0,C 180,E1 -5129.221,E2 -5129.221} C_VEL
LIN {X 0,Y 516.157,Z 634.228,A -85,B 0,C 180,E1 -5130.781,E2 -5130.781} C_VEL
LIN {X 0,Y 516.259,Z 632.892,A -85,B 0,C 180,E1 -5132.342,E2 -5132.342} C_VEL
LIN {X 0,Y 516.325,Z 630.198,A -85,B 0,C 180,E1 -5133.904,E2 -5133.904} C_VEL
LIN {X 0,Y 516.386,Z 626.072,A -85,B 0,C 180,E1 -5135.468,E2 -5135.468} C_VEL
LIN {X 0,Y 516.404,Z 620.383,A -85,B 0,C 180,E1 -5137.037,E2 -5137.037} C_VEL
LIN {X 0,Y 516.583,Z 613.966,A -85,B 0,C 180,E1 -5138.411,E2 -5138.411} C_VEL
LIN {X 0,Y 516.809,Z 605.996,A -85,B 0,C 180,E1 -5139.788,E2 -5139.788} C_VEL
LIN {X 0,Y 517.103,Z 597.658,A -85,B 0,C 180,E1 -5140.97,E2 -5140.97} C_VEL
LIN {X 0,Y 517.455,Z 587.22,A -85,B 0,C 180,E1 -5142.198,E2 -5142.198} C_VEL
LIN {X 0,Y 517.827,Z 576.418,A -85,B 0,C 180,E1 -5143.241,E2 -5143.241} C_VEL
LIN {X 0,Y 518.263,Z 563.845,A -85,B 0,C 180,E1 -5144.229,E2 -5144.229} C_VEL
LIN {X 0,Y 518.701,Z 551.368,A -85,B 0,C 180,E1 -5145.019,E2 -5145.019} C_VEL
LIN {X 0,Y 519.09,Z 538.549,A -85,B 0,C 180,E1 -5145.661,E2 -5145.661} C_VEL
LIN {X 0,Y 519.387,Z 524.679,A -85,B 0,C 180,E1 -5146.187,E2 -5146.187} C_VEL
LIN {X 0,Y 519.656,Z 510.701,A -85,B 0,C 180,E1 -5146.551,E2 -5146.551} C_VEL
LIN {X 0,Y 519.888,Z 482.58,A -85,B 0,C 180,E1 -5146.973,E2 -5146.973} C_VEL
LIN {X 0,Y 520.297,Z 384.012,A -85,B 0,C 180,E1 -5148.358,E2 -5148.358} C_VEL
LIN {X 0,Y 517.985,Z 371.554,A -85,B 0,C 180,E1 -5148.635,E2 -5148.635} C_VEL
LIN {X 0,Y 518.539,Z 351.634,A -85,B 0,C 180,E1 -5151.675,E2 -5151.675} C_VEL
LIN {X 0,Y 518.852,Z 339.517,A -85,B 0,C 180,E1 -5153.553,E2 -5153.553} C_VEL
LIN {X 0,Y 516.869,Z 329.729,A -85,B 0,C 180,E1 -5155.227,E2 -5155.227} C_VEL
LIN {X 0,Y 516.844,Z 329.728,A -85,B 0,C 180,E1 -5158.421,E2 -5158.421} C_VEL
LIN {X 0,Y 516.89,Z 329.725,A -85,B 0,C 180,E1 -5161.11,E2 -5161.11} C_VEL
LIN {X 0,Y 516.912,Z 329.719,A -85,B 0,C 180,E1 -5163.966,E2 -5163.966} C_VEL
LIN {X 0,Y 516.858,Z 329.727,A -85,B 0,C 180,E1 -5166.749,E2 -5166.749} C_VEL
LIN {X 0,Y 516.887,Z 329.721,A -85,B 0,C 180,E1 -5169.722,E2 -5169.722} C_VEL
LIN {X 0,Y 516.916,Z 329.717,A -85,B 0,C 180,E1 -5171.776,E2 -5171.776} C_VEL
LIN {X 0,Y 516.928,Z 329.722,A -85,B 0,C 180,E1 -5175.011,E2 -5175.011} C_VEL
LIN {X 0,Y 516.918,Z 329.721,A -85,B 0,C 180,E1 -5178.399,E2 -5178.399} C_VEL
LIN {X 0,Y 516.884,Z 329.722,A -85,B 0,C 180,E1 -5181.284,E2 -5181.284} C_VEL
LIN {X 0,Y 516.872,Z 329.728,A -85,B 0,C 180,E1 -5184.22,E2 -5184.22} C_VEL
LIN {X 0,Y 516.9,Z 329.721,A -85,B 0,C 180,E1 -5187.053,E2 -5187.053} C_VEL
LIN {X 0,Y 516.896,Z 329.725,A -85,B 0,C 180,E1 -5189.797,E2 -5189.797} C_VEL
LIN {X 0,Y 516.891,Z 329.727,A -85,B 0,C 180,E1 -5192.465,E2 -5192.465} C_VEL
LIN {X 0,Y 516.877,Z 329.729,A -85,B 0,C 180,E1 -5195.646,E2 -5195.646} C_VEL
LIN {X 0,Y 516.926,Z 329.783,A -85,B 0,C 180,E1 -5197.458,E2 -5197.458} C_VEL
LIN {X 0,Y 517.965,Z 336.171,A -85,B 0,C 180,E1 -5198.509,E2 -5198.509} C_VEL
LIN {X 0,Y 517.786,Z 352.876,A -85,B 0,C 180,E1 -5201.194,E2 -5201.194} C_VEL
LIN {X 0,Y 517.544,Z 370.441,A -85,B 0,C 180,E1 -5204.039,E2 -5204.039} C_VEL
LIN {X 0,Y 517.463,Z 374.546,A -85,B 0,C 180,E1 -5204.713,E2 -5204.713} C_VEL
LIN {X 0,Y 519.072,Z 384.615,A -85,B 0,C 180,E1 -5204.921,E2 -5204.921} C_VEL
LIN {X 0,Y 518.467,Z 482.974,A -85,B 0,C 180,E1 -5206.378,E2 -5206.378} C_VEL
LIN {X 0,Y 518.294,Z 495.962,A -85,B 0,C 180,E1 -5206.722,E2 -5206.722} C_VEL
LIN {X 0,Y 518.065,Z 508.362,A -85,B 0,C 180,E1 -5207.215,E2 -5207.215} C_VEL
LIN {X 0,Y 517.802,Z 520.705,A -85,B 0,C 180,E1 -5207.874,E2 -5207.874} C_VEL
LIN {X 0,Y 517.575,Z 531.816,A -85,B 0,C 180,E1 -5208.645,E2 -5208.645} C_VEL
LIN {X 0,Y 517.246,Z 542.047,A -85,B 0,C 180,E1 -5209.529,E2 -5209.529} C_VEL
LIN {X 0,Y 517.032,Z 550.457,A -85,B 0,C 180,E1 -5210.415,E2 -5210.415} C_VEL
LIN {X 0,Y 516.816,Z 558.178,A -85,B 0,C 180,E1 -5211.397,E2 -5211.397} C_VEL
LIN {X 0,Y 516.595,Z 565.727,A -85,B 0,C 180,E1 -5212.574,E2 -5212.574} C_VEL
LIN {X 0,Y 516.494,Z 571.753,A -85,B 0,C 180,E1 -5213.751,E2 -5213.751} C_VEL
LIN {X 0,Y 516.321,Z 576.527,A -85,B 0,C 180,E1 -5214.924,E2 -5214.924} C_VEL
LIN {X 0,Y 516.374,Z 580.14,A -85,B 0,C 180,E1 -5216.098,E2 -5216.098} C_VEL
LIN {X 0,Y 516.351,Z 582.018,A -85,B 0,C 180,E1 -5216.879,E2 -5216.879} C_VEL
LIN {X 0,Y 516.263,Z 583.45,A -85,B 0,C 180,E1 -5217.659,E2 -5217.659} C_VEL
LIN {X 0,Y 516.163,Z 585.095,A -85,B 0,C 180,E1 -5219.22,E2 -5219.22} C_VEL
LIN {X 0,Y 516.161,Z 585.319,A -85,B 0,C 180,E1 -5220,E2 -5220} C_VEL
LIN {X 0,Y 516.163,Z 585.136,A -85,B 0,C 180,E1 -5220.78,E2 -5220.78} C_VEL
LIN {X 0,Y 516.192,Z 584.541,A -85,B 0,C 180,E1 -5221.56,E2 -5221.56} C_VEL
LIN {X 0,Y 516.31,Z 582.156,A -85,B 0,C 180,E1 -5223.121,E2 -5223.121} C_VEL
LIN {X 0,Y 516.366,Z 579.281,A -85,B 0,C 180,E1 -5224.293,E2 -5224.293} C_VEL
LIN {X 0,Y 516.405,Z 575.338,A -85,B 0,C 180,E1 -5225.467,E2 -5225.467} C_VEL
LIN {X 0,Y 516.512,Z 570.274,A -85,B 0,C 180,E1 -5226.639,E2 -5226.639} C_VEL
LIN {X 0,Y 516.644,Z 563.84,A -85,B 0,C 180,E1 -5227.818,E2 -5227.818} C_VEL
LIN {X 0,Y 516.862,Z 555.861,A -85,B 0,C 180,E1 -5228.996,E2 -5228.996} C_VEL
LIN {X 0,Y 517.082,Z 547.662,A -85,B 0,C 180,E1 -5229.979,E2 -5229.979} C_VEL
LIN {X 0,Y 517.36,Z 537.619,A -85,B 0,C 180,E1 -5230.963,E2 -5230.963} C_VEL
LIN {X 0,Y 517.674,Z 527.691,A -85,B 0,C 180,E1 -5231.75,E2 -5231.75} C_VEL
LIN {X 0,Y 517.912,Z 516.331,A -85,B 0,C 180,E1 -5232.476,E2 -5232.476} C_VEL
LIN {X 0,Y 518.146,Z 503.875,A -85,B 0,C 180,E1 -5233.082,E2 -5233.082} C_VEL
LIN {X 0,Y 518.409,Z 490.463,A -85,B 0,C 180,E1 -5233.549,E2 -5233.549} C_VEL
LIN {X 0,Y 518.563,Z 476.68,A -85,B 0,C 180,E1 -5233.845,E2 -5233.845} C_VEL
LIN {X 0,Y 518.961,Z 382.997,A -85,B 0,C 180,E1 -5235.2,E2 -5235.2} C_VEL
LIN {X 0,Y 517.414,Z 373.956,A -85,B 0,C 180,E1 -5235.402,E2 -5235.402} C_VEL
LIN {X 0,Y 517.73,Z 355.936,A -85,B 0,C 180,E1 -5238.398,E2 -5238.398} C_VEL
LIN {X 0,Y 518.033,Z 338.667,A -85,B 0,C 180,E1 -5241.279,E2 -5241.279} C_VEL
LIN {X 0,Y 517.655,Z 333.672,A -85,B 0,C 180,E1 -5242.133,E2 -5242.133} C_VEL
LIN {X 0,Y 516.896,Z 329.725,A -85,B 0,C 180,E1 -5242.858,E2 -5242.858} C_VEL
LIN {X 0,Y 516.946,Z 329.721,A -85,B 0,C 180,E1 -5246.195,E2 -5246.195} C_VEL
LIN {X 0,Y 516.926,Z 329.715,A -85,B 0,C 180,E1 -5249.304,E2 -5249.304} C_VEL
LIN {X 0,Y 516.901,Z 329.721,A -85,B 0,C 180,E1 -5252.543,E2 -5252.543} C_VEL
LIN {X 0,Y 516.877,Z 329.721,A -85,B 0,C 180,E1 -5254.986,E2 -5254.986} C_VEL
LIN {X 0,Y 516.204,Z 329.811,A -85,B 0,C 180,E1 -5255.636,E2 -5255.636} C_VEL
LIN {X 0,Y 513.381,Z 330.162,A -85,B 0,C 180,E1 -5256.692,E2 -5256.692} C_VEL
LIN {X 0,Y 510.989,Z 330.461,A -85,B 0,C 180,E1 -5257.543,E2 -5257.543} C_VEL
LIN {X 0,Y 509.942,Z 330.59,A -85,B 0,C 180,E1 -5258.2,E2 -5258.2} C_VEL
LIN {X 0,Y 509.846,Z 330.599,A -85,B 0,C 180,E1 -5258.422,E2 -5258.422} C_VEL
LIN {X 0,Y 509.849,Z 330.6,A -85,B 0,C 180,E1 -5261.426,E2 -5261.426} C_VEL
LIN {X 0,Y 509.844,Z 330.598,A -85,B 0,C 180,E1 -5264.67,E2 -5264.67} C_VEL
LIN {X 0,Y 509.807,Z 330.609,A -85,B 0,C 180,E1 -5267.506,E2 -5267.506} C_VEL
LIN {X 0,Y 509.836,Z 330.599,A -85,B 0,C 180,E1 -5270.646,E2 -5270.646} C_VEL
LIN {X 0,Y 509.808,Z 330.609,A -85,B 0,C 180,E1 -5273.644,E2 -5273.644} C_VEL
LIN {X 0,Y 509.829,Z 330.601,A -85,B 0,C 180,E1 -5276.536,E2 -5276.536} C_VEL
LIN {X 0,Y 509.809,Z 330.608,A -85,B 0,C 180,E1 -5279.331,E2 -5279.331} C_VEL
LIN {X 0,Y 509.829,Z 330.601,A -85,B 0,C 180,E1 -5282.05,E2 -5282.05} C_VEL
LIN {X 0,Y 509.782,Z 330.611,A -85,B 0,C 180,E1 -5284.698,E2 -5284.698} C_VEL
LIN {X 0,Y 509.834,Z 330.721,A -85,B 0,C 180,E1 -5285.761,E2 -5285.761} C_VEL
LIN {X 0,Y 511.64,Z 339.744,A -85,B 0,C 180,E1 -5287.379,E2 -5287.379} C_VEL
LIN {X 0,Y 511.388,Z 352.702,A -85,B 0,C 180,E1 -5289.529,E2 -5289.529} C_VEL
LIN {X 0,Y 511.032,Z 362.737,A -85,B 0,C 180,E1 -5291.164,E2 -5291.164} C_VEL
LIN {X 0,Y 513.68,Z 376.278,A -85,B 0,C 180,E1 -5291.465,E2 -5291.465} C_VEL
LIN {X 0,Y 512.879,Z 499.271,A -85,B 0,C 180,E1 -5293.224,E2 -5293.224} C_VEL
LIN {X 0,Y 512.607,Z 513.493,A -85,B 0,C 180,E1 -5293.578,E2 -5293.578} C_VEL
LIN {X 0,Y 512.328,Z 527.023,A -85,B 0,C 180,E1 -5294.075,E2 -5294.075} C_VEL
LIN {X 0,Y 511.952,Z 539.401,A -85,B 0,C 180,E1 -5294.676,E2 -5294.676} C_VEL
LIN {X 0,Y 511.449,Z 552.339,A -85,B 0,C 180,E1 -5295.475,E2 -5295.475} C_VEL
LIN {X 0,Y 511.017,Z 564.071,A -85,B 0,C 180,E1 -5296.377,E2 -5296.377} C_VEL
LIN {X 0,Y 510.556,Z 575.689,A -85,B 0,C 180,E1 -5297.469,E2 -5297.469} C_VEL
LIN {X 0,Y 510.205,Z 586.225,A -85,B 0,C 180,E1 -5298.679,E2 -5298.679} C_VEL
LIN {X 0,Y 509.832,Z 594.848,A -85,B 0,C 180,E1 -5299.876,E2 -5299.876} C_VEL
LIN {X 0,Y 509.605,Z 603.114,A -85,B 0,C 180,E1 -5301.273,E2 -5301.273} C_VEL
LIN {X 0,Y 509.414,Z 608.875,A -85,B 0,C 180,E1 -5302.468,E2 -5302.468} C_VEL
LIN {X 0,Y 509.309,Z 613.617,A -85,B 0,C 180,E1 -5303.661,E2 -5303.661} C_VEL
LIN {X 0,Y 509.238,Z 617.46,A -85,B 0,C 180,E1 -5304.852,E2 -5304.852} C_VEL
LIN {X 0,Y 509.251,Z 620.405,A -85,B 0,C 180,E1 -5306.042,E2 -5306.042} C_VEL
LIN {X 0,Y 509.189,Z 623.129,A -85,B 0,C 180,E1 -5307.626,E2 -5307.626} C_VEL
LIN {X 0,Y 509.07,Z 624.484,A -85,B 0,C 180,E1 -5309.208,E2 -5309.208} C_VEL
LIN {X 0,Y 509.071,Z 624.515,A -85,B 0,C 180,E1 -5310.79,E2 -5310.79} C_VEL
LIN {X 0,Y 509.188,Z 623.252,A -85,B 0,C 180,E1 -5312.372,E2 -5312.372} C_VEL
LIN {X 0,Y 509.25,Z 620.616,A -85,B 0,C 180,E1 -5313.956,E2 -5313.956} C_VEL
LIN {X 0,Y 509.315,Z 616.54,A -85,B 0,C 180,E1 -5315.542,E2 -5315.542} C_VEL
LIN {X 0,Y 509.362,Z 610.927,A -85,B 0,C 180,E1 -5317.132,E2 -5317.132} C_VEL
LIN {X 0,Y 509.556,Z 604.59,A -85,B 0,C 180,E1 -5318.525,E2 -5318.525} C_VEL
LIN {X 0,Y 509.791,Z 596.704,A -85,B 0,C 180,E1 -5319.922,E2 -5319.922} C_VEL
LIN {X 0,Y 510.101,Z 588.455,A -85,B 0,C 180,E1 -5321.12,E2 -5321.12} C_VEL
LIN {X 0,Y 510.455,Z 578.795,A -85,B 0,C 180,E1 -5322.289,E2 -5322.289} C_VEL
LIN {X 0,Y 510.893,Z 567.457,A -85,B 0,C 180,E1 -5323.422,E2 -5323.422} C_VEL
LIN {X 0,Y 511.305,Z 556.451,A -85,B 0,C 180,E1 -5324.323,E2 -5324.323} C_VEL
LIN {X 0,Y 511.76,Z 544.508,A -85,B 0,C 180,E1 -5325.124,E2 -5325.124} C_VEL
LIN {X 0,Y 512.206,Z 531.313,A -85,B 0,C 180,E1 -5325.824,E2 -5325.824} C_VEL
LIN {X 0,Y 512.574,Z 517.447,A -85,B 0,C 180,E1 -5326.38,E2 -5326.38} C_VEL
LIN {X 0,Y 512.818,Z 503.435,A -85,B 0,C 180,E1 -5326.776,E2 -5326.776} C_VEL
LIN {X 0,Y 513.014,Z 485.474,A -85,B 0,C 180,E1 -5327.077,E2 -5327.077} C_VEL
LIN {X 0,Y 513.718,Z 376.617,A -85,B 0,C 180,E1 -5328.619,E2 -5328.619} C_VEL
LIN {X 0,Y 511.025,Z 362.734,A -85,B 0,C 180,E1 -5328.927,E2 -5328.927} C_VEL
LIN {X 0,Y 511.624,Z 345.373,A -85,B 0,C 180,E1 -5331.769,E2 -5331.769} C_VEL
LIN {X 0,Y 511.565,Z 339.098,A -85,B 0,C 180,E1 -5332.823,E2 -5332.823} C_VEL
LIN {X 0,Y 509.847,Z 330.605,A -85,B 0,C 180,E1 -5334.371,E2 -5334.371} C_VEL
LIN {X 0,Y 509.814,Z 330.609,A -85,B 0,C 180,E1 -5337.058,E2 -5337.058} C_VEL
LIN {X 0,Y 509.82,Z 330.604,A -85,B 0,C 180,E1 -5339.752,E2 -5339.752} C_VEL
LIN {X 0,Y 509.859,Z 330.604,A -85,B 0,C 180,E1 -5342.771,E2 -5342.771} C_VEL
LIN {X 0,Y 509.815,Z 330.603,A -85,B 0,C 180,E1 -5345.576,E2 -5345.576} C_VEL
LIN {X 0,Y 509.812,Z 330.603,A -85,B 0,C 180,E1 -5348.339,E2 -5348.339} C_VEL
LIN {X 0,Y 509.795,Z 330.605,A -85,B 0,C 180,E1 -5351.429,E2 -5351.429} C_VEL
LIN {X 0,Y 509.829,Z 330.605,A -85,B 0,C 180,E1 -5354.669,E2 -5354.669} C_VEL
LIN {X 0,Y 509.791,Z 330.605,A -85,B 0,C 180,E1 -5357.506,E2 -5357.506} C_VEL
LIN {X 0,Y 509.824,Z 330.606,A -85,B 0,C 180,E1 -5360.645,E2 -5360.645} C_VEL
LIN {X 0,Y 509.796,Z 330.603,A -85,B 0,C 180,E1 -5363.644,E2 -5363.644} C_VEL
LIN {X 0,Y 509.825,Z 330.603,A -85,B 0,C 180,E1 -5366.536,E2 -5366.536} C_VEL
LIN {X 0,Y 509.814,Z 330.602,A -85,B 0,C 180,E1 -5369.332,E2 -5369.332} C_VEL
LIN {X 0,Y 509.818,Z 330.599,A -85,B 0,C 180,E1 -5372.05,E2 -5372.05} C_VEL
LIN {X 0,Y 509.788,Z 330.605,A -85,B 0,C 180,E1 -5374.699,E2 -5374.699} C_VEL
LIN {X 0,Y 509.81,Z 330.602,A -85,B 0,C 180,E1 -5377.458,E2 -5377.458} C_VEL
LIN {X 0,Y 509.893,Z 330.586,A -85,B 0,C 180,E1 -5379.844,E2 -5379.844} C_VEL
LIN {X 0,Y 509.836,Z 330.6,A -85,B 0,C 180,E1 -5383.173,E2 -5383.173} C_VEL
LIN {X 0,Y 509.827,Z 330.599,A -85,B 0,C 180,E1 -5385.633,E2 -5385.633} C_VEL
LIN {X 0,Y 509.891,Z 330.596,A -85,B 0,C 180,E1 -5388.874,E2 -5388.874} C_VEL
LIN {X 0,Y 509.891,Z 330.592,A -85,B 0,C 180,E1 -5392.077,E2 -5392.077} C_VEL
LIN {X 0,Y 509.917,Z 330.595,A -85,B 0,C 180,E1 -5394.464,E2 -5394.464} C_VEL
LIN {X 0,Y 510.026,Z 330.574,A -85,B 0,C 180,E1 -5397.631,E2 -5397.631} C_VEL
LIN {X 0,Y 510.044,Z 330.577,A -85,B 0,C 180,E1 -5400.789,E2 -5400.789} C_VEL
LIN {X 0,Y 509.894,Z 330.591,A -85,B 0,C 180,E1 -5403.16,E2 -5403.16} C_VEL
LIN {X 0,Y 509.902,Z 330.595,A -85,B 0,C 180,E1 -5406.33,E2 -5406.33} C_VEL
LIN {X 0,Y 509.835,Z 330.597,A -85,B 0,C 180,E1 -5409.521,E2 -5409.521} C_VEL
LIN {X 0,Y 509.884,Z 330.593,A -85,B 0,C 180,E1 -5411.932,E2 -5411.932} C_VEL
LIN {X 0,Y 509.879,Z 330.593,A -85,B 0,C 180,E1 -5415.242,E2 -5415.242} C_VEL
LIN {X 0,Y 509.822,Z 330.608,A -85,B 0,C 180,E1 -5418.485,E2 -5418.485} C_VEL
LIN {X 0,Y 509.835,Z 330.595,A -85,B 0,C 180,E1 -5421.002,E2 -5421.002} C_VEL
LIN {X 0,Y 509.803,Z 330.598,A -85,B 0,C 180,E1 -5423.565,E2 -5423.565} C_VEL
LIN {X 0,Y 509.793,Z 330.612,A -85,B 0,C 180,E1 -5426.355,E2 -5426.355} C_VEL
LIN {X 0,Y 509.834,Z 330.596,A -85,B 0,C 180,E1 -5428.847,E2 -5428.847} C_VEL
LIN {X 0,Y 509.797,Z 330.603,A -85,B 0,C 180,E1 -5431.592,E2 -5431.592} C_VEL
LIN {X 0,Y 509.819,Z 330.608,A -85,B 0,C 180,E1 -5434.416,E2 -5434.416} C_VEL
LIN {X 0,Y 509.766,Z 330.607,A -85,B 0,C 180,E1 -5437.345,E2 -5437.345} C_VEL
LIN {X 0,Y 509.774,Z 330.612,A -85,B 0,C 180,E1 -5440.388,E2 -5440.388} C_VEL
LIN {X 0,Y 509.78,Z 330.606,A -85,B 0,C 180,E1 -5443.576,E2 -5443.576} C_VEL
LIN {X 0,Y 509.779,Z 330.612,A -85,B 0,C 180,E1 -5446.426,E2 -5446.426} C_VEL
LIN {X 0,Y 509.775,Z 330.608,A -85,B 0,C 180,E1 -5449.614,E2 -5449.614} C_VEL
LIN {X 0,Y 509.766,Z 330.611,A -85,B 0,C 180,E1 -5452.657,E2 -5452.657} C_VEL
LIN {X 0,Y 509.83,Z 330.604,A -85,B 0,C 180,E1 -5455.802,E2 -5455.802} C_VEL
LIN {X 0,Y 509.829,Z 330.601,A -85,B 0,C 180,E1 -5458.723,E2 -5458.723} C_VEL
LIN {X 0,Y 509.826,Z 330.6,A -85,B 0,C 180,E1 -5461.154,E2 -5461.154} C_VEL
LIN {X 0,Y 509.821,Z 330.608,A -85,B 0,C 180,E1 -5464.265,E2 -5464.265} C_VEL
LIN {X 0,Y 509.817,Z 330.704,A -85,B 0,C 180,E1 -5464.593,E2 -5464.593} C_VEL
LIN {X 0,Y 511.953,Z 340.823,A -85,B 0,C 180,E1 -5466.327,E2 -5466.327} C_VEL
LIN {X 0,Y 511.61,Z 354.286,A -85,B 0,C 180,E1 -5468.442,E2 -5468.442} C_VEL
LIN {X 0,Y 511.03,Z 371.573,A -85,B 0,C 180,E1 -5471.115,E2 -5471.115} C_VEL
LIN {X 0,Y 513.697,Z 386.408,A -85,B 0,C 180,E1 -5471.433,E2 -5471.433} C_VEL
LIN {X 0,Y 512.86,Z 509.6,A -85,B 0,C 180,E1 -5473.2,E2 -5473.2} C_VEL
LIN {X 0,Y 512.567,Z 524.148,A -85,B 0,C 180,E1 -5473.577,E2 -5473.577} C_VEL
LIN {X 0,Y 512.224,Z 537.394,A -85,B 0,C 180,E1 -5474.075,E2 -5474.075} C_VEL
LIN {X 0,Y 511.832,Z 551.344,A -85,B 0,C 180,E1 -5474.777,E2 -5474.777} C_VEL
LIN {X 0,Y 511.346,Z 563.814,A -85,B 0,C 180,E1 -5475.576,E2 -5475.576} C_VEL
LIN {X 0,Y 510.84,Z 576.376,A -85,B 0,C 180,E1 -5476.577,E2 -5476.577} C_VEL
LIN {X 0,Y 510.444,Z 587.776,A -85,B 0,C 180,E1 -5477.702,E2 -5477.702} C_VEL
LIN {X 0,Y 510.09,Z 597.608,A -85,B 0,C 180,E1 -5478.88,E2 -5478.88} C_VEL
LIN {X 0,Y 509.744,Z 605.943,A -85,B 0,C 180,E1 -5480.077,E2 -5480.077} C_VEL
LIN {X 0,Y 509.539,Z 613.912,A -85,B 0,C 180,E1 -5481.474,E2 -5481.474} C_VEL
LIN {X 0,Y 509.326,Z 620.324,A -85,B 0,C 180,E1 -5482.867,E2 -5482.867} C_VEL
LIN {X 0,Y 509.299,Z 626.012,A -85,B 0,C 180,E1 -5484.458,E2 -5484.458} C_VEL
LIN {X 0,Y 509.218,Z 630.14,A -85,B 0,C 180,E1 -5486.044,E2 -5486.044} C_VEL
LIN {X 0,Y 509.159,Z 632.831,A -85,B 0,C 180,E1 -5487.628,E2 -5487.628} C_VEL
LIN {X 0,Y 509.071,Z 634.162,A -85,B 0,C 180,E1 -5489.21,E2 -5489.21} C_VEL
LIN {X 0,Y 509.071,Z 634.161,A -85,B 0,C 180,E1 -5490.792,E2 -5490.792} C_VEL
LIN {X 0,Y 509.159,Z 632.825,A -85,B 0,C 180,E1 -5492.374,E2 -5492.374} C_VEL
LIN {X 0,Y 509.218,Z 630.13,A -85,B 0,C 180,E1 -5493.958,E2 -5493.958} C_VEL
LIN {X 0,Y 509.297,Z 626.004,A -85,B 0,C 180,E1 -5495.544,E2 -5495.544} C_VEL
LIN {X 0,Y 509.329,Z 620.316,A -85,B 0,C 180,E1 -5497.135,E2 -5497.135} C_VEL
LIN {X 0,Y 509.541,Z 613.899,A -85,B 0,C 180,E1 -5498.528,E2 -5498.528} C_VEL
LIN {X 0,Y 509.749,Z 605.928,A -85,B 0,C 180,E1 -5499.925,E2 -5499.925} C_VEL
LIN {X 0,Y 510.112,Z 597.59,A -85,B 0,C 180,E1 -5501.122,E2 -5501.122} C_VEL
LIN {X 0,Y 510.451,Z 587.5,A -85,B 0,C 180,E1 -5502.329,E2 -5502.329} C_VEL
LIN {X 0,Y 510.891,Z 576.35,A -85,B 0,C 180,E1 -5503.424,E2 -5503.424} C_VEL
LIN {X 0,Y 511.317,Z 565.203,A -85,B 0,C 180,E1 -5504.325,E2 -5504.325} C_VEL
LIN {X 0,Y 511.749,Z 553.067,A -85,B 0,C 180,E1 -5505.126,E2 -5505.126} C_VEL
LIN {X 0,Y 512.219,Z 539.612,A -85,B 0,C 180,E1 -5505.826,E2 -5505.826} C_VEL
LIN {X 0,Y 512.54,Z 525.226,A -85,B 0,C 180,E1 -5506.388,E2 -5506.388} C_VEL
LIN {X 0,Y 512.862,Z 510.634,A -85,B 0,C 180,E1 -5506.777,E2 -5506.777} C_VEL
LIN {X 0,Y 513.091,Z 484.302,A -85,B 0,C 180,E1 -5507.18,E2 -5507.18} C_VEL
LIN {X 0,Y 513.591,Z 385.211,A -85,B 0,C 180,E1 -5508.588,E2 -5508.588} C_VEL
LIN {X 0,Y 511.053,Z 371.415,A -85,B 0,C 180,E1 -5508.908,E2 -5508.908} C_VEL
LIN {X 0,Y 511.627,Z 352.924,A -85,B 0,C 180,E1 -5511.771,E2 -5511.771} C_VEL
LIN {X 0,Y 512.063,Z 342.152,A -85,B 0,C 180,E1 -5513.456,E2 -5513.456} C_VEL
LIN {X 0,Y 509.985,Z 331.358,A -85,B 0,C 180,E1 -5515.291,E2 -5515.291} C_VEL
LIN {X 0,Y 509.815,Z 330.609,A -85,B 0,C 180,E1 -5515.464,E2 -5515.464} C_VEL
LIN {X 0,Y 509.813,Z 330.606,A -85,B 0,C 180,E1 -5518.083,E2 -5518.083} C_VEL
LIN {X 0,Y 509.837,Z 330.601,A -85,B 0,C 180,E1 -5520.667,E2 -5520.667} C_VEL
LIN {X 0,Y 509.863,Z 330.602,A -85,B 0,C 180,E1 -5523.462,E2 -5523.462} C_VEL
LIN {X 0,Y 509.814,Z 330.602,A -85,B 0,C 180,E1 -5526.355,E2 -5526.355} C_VEL
LIN {X 0,Y 509.851,Z 330.601,A -85,B 0,C 180,E1 -5529.353,E2 -5529.353} C_VEL
LIN {X 0,Y 509.838,Z 330.601,A -85,B 0,C 180,E1 -5532.49,E2 -5532.49} C_VEL
LIN {X 0,Y 509.862,Z 330.598,A -85,B 0,C 180,E1 -5535.333,E2 -5535.333} C_VEL
LIN {X 0,Y 509.86,Z 330.601,A -85,B 0,C 180,E1 -5538.575,E2 -5538.575} C_VEL
LIN {X 0,Y 509.854,Z 330.597,A -85,B 0,C 180,E1 -5541.787,E2 -5541.787} C_VEL
LIN {X 0,Y 509.832,Z 330.604,A -85,B 0,C 180,E1 -5544.622,E2 -5544.622} C_VEL
LIN {X 0,Y 509.866,Z 330.597,A -85,B 0,C 180,E1 -5547.481,E2 -5547.481} C_VEL
LIN {X 0,Y 509.863,Z 330.604,A -85,B 0,C 180,E1 -5550.274,E2 -5550.274} C_VEL
LIN {X 0,Y 509.832,Z 330.604,A -85,B 0,C 180,E1 -5552.941,E2 -5552.941} C_VEL
LIN {X 0,Y 509.839,Z 330.605,A -85,B 0,C 180,E1 -5555.572,E2 -5555.572} C_VEL
LIN {X 0,Y 509.893,Z 330.645,A -85,B 0,C 180,E1 -5557.298,E2 -5557.298} C_VEL
LIN {X 0,Y 511.009,Z 337.391,A -85,B 0,C 180,E1 -5558.414,E2 -5558.414} C_VEL
LIN {X 0,Y 510.843,Z 354.297,A -85,B 0,C 180,E1 -5561.137,E2 -5561.137} C_VEL
LIN {X 0,Y 510.558,Z 373.953,A -85,B 0,C 180,E1 -5564.344,E2 -5564.344} C_VEL
LIN {X 0,Y 510.535,Z 374.892,A -85,B 0,C 180,E1 -5564.499,E2 -5564.499} C_VEL
LIN {X 0,Y 512.215,Z 384.741,A -85,B 0,C 180,E1 -5564.719,E2 -5564.719} C_VEL
LIN {X 0,Y 511.547,Z 483.288,A -85,B 0,C 180,E1 -5566.215,E2 -5566.215} C_VEL
LIN {X 0,Y 511.366,Z 495.506,A -85,B 0,C 180,E1 -5566.539,E2 -5566.539} C_VEL
LIN {X 0,Y 511.105,Z 508.155,A -85,B 0,C 180,E1 -5567.038,E2 -5567.038} C_VEL
LIN {X 0,Y 510.852,Z 520.598,A -85,B 0,C 180,E1 -5567.705,E2 -5567.705} C_VEL
LIN {X 0,Y 510.605,Z 531.854,A -85,B 0,C 180,E1 -5568.488,E2 -5568.488} C_VEL
LIN {X 0,Y 510.22,Z 543.196,A -85,B 0,C 180,E1 -5569.484,E2 -5569.484} C_VEL
LIN {X 0,Y 509.949,Z 552.306,A -85,B 0,C 180,E1 -5570.481,E2 -5570.481} C_VEL
LIN {X 0,Y 509.678,Z 561.087,A -85,B 0,C 180,E1 -5571.675,E2 -5571.675} C_VEL
LIN {X 0,Y 509.527,Z 568.15,A -85,B 0,C 180,E1 -5572.869,E2 -5572.869} C_VEL
LIN {X 0,Y 509.431,Z 573.772,A -85,B 0,C 180,E1 -5574.061,E2 -5574.061} C_VEL
LIN {X 0,Y 509.225,Z 578.164,A -85,B 0,C 180,E1 -5575.25,E2 -5575.25} C_VEL
LIN {X 0,Y 509.306,Z 580.454,A -85,B 0,C 180,E1 -5576.044,E2 -5576.044} C_VEL
LIN {X 0,Y 509.263,Z 582.34,A -85,B 0,C 180,E1 -5576.836,E2 -5576.836} C_VEL
LIN {X 0,Y 509.194,Z 583.778,A -85,B 0,C 180,E1 -5577.627,E2 -5577.627} C_VEL
LIN {X 0,Y 509.077,Z 585.413,A -85,B 0,C 180,E1 -5579.209,E2 -5579.209} C_VEL
LIN {X 0,Y 509.072,Z 585.642,A -85,B 0,C 180,E1 -5580,E2 -5580} C_VEL
LIN {X 0,Y 509.077,Z 585.453,A -85,B 0,C 180,E1 -5580.791,E2 -5580.791} C_VEL
LIN {X 0,Y 509.192,Z 583.854,A -85,B 0,C 180,E1 -5582.373,E2 -5582.373} C_VEL
LIN {X 0,Y 509.227,Z 582.463,A -85,B 0,C 180,E1 -5583.165,E2 -5583.165} C_VEL
LIN {X 0,Y 509.29,Z 579.563,A -85,B 0,C 180,E1 -5584.353,E2 -5584.353} C_VEL
LIN {X 0,Y 509.348,Z 575.599,A -85,B 0,C 180,E1 -5585.543,E2 -5585.543} C_VEL
LIN {X 0,Y 509.444,Z 569.687,A -85,B 0,C 180,E1 -5586.896,E2 -5586.896} C_VEL
LIN {X 0,Y 509.632,Z 562.828,A -85,B 0,C 180,E1 -5588.126,E2 -5588.126} C_VEL
LIN {X 0,Y 509.864,Z 554.485,A -85,B 0,C 180,E1 -5589.321,E2 -5589.321} C_VEL
LIN {X 0,Y 510.093,Z 545.915,A -85,B 0,C 180,E1 -5590.318,E2 -5590.318} C_VEL
LIN {X 0,Y 510.465,Z 535.392,A -85,B 0,C 180,E1 -5591.314,E2 -5591.314} C_VEL
LIN {X 0,Y 510.76,Z 524.405,A -85,B 0,C 180,E1 -5592.143,E2 -5592.143} C_VEL
LIN {X 0,Y 511.035,Z 513.196,A -85,B 0,C 180,E1 -5592.812,E2 -5592.812} C_VEL
LIN {X 0,Y 511.322,Z 501.236,A -85,B 0,C 180,E1 -5593.361,E2 -5593.361} C_VEL
LIN {X 0,Y 511.527,Z 488.057,A -85,B 0,C 180,E1 -5593.786,E2 -5593.786} C_VEL
LIN {X 0,Y 511.661,Z 473.979,A -85,B 0,C 180,E1 -5594.061,E2 -5594.061} C_VEL
LIN {X 0,Y 512.129,Z 384.014,A -85,B 0,C 180,E1 -5595.392,E2 -5595.392} C_VEL
LIN {X 0,Y 510.474,Z 374.267,A -85,B 0,C 180,E1 -5595.6,E2 -5595.6} C_VEL
LIN {X 0,Y 510.795,Z 355.991,A -85,B 0,C 180,E1 -5598.657,E2 -5598.657} C_VEL
LIN {X 0,Y 511.089,Z 338.529,A -85,B 0,C 180,E1 -5601.583,E2 -5601.583} C_VEL
LIN {X 0,Y 509.941,Z 330.98,A -85,B 0,C 180,E1 -5602.914,E2 -5602.914} C_VEL
LIN {X 0,Y 509.851,Z 330.602,A -85,B 0,C 180,E1 -5603.025,E2 -5603.025} C_VEL
LIN {X 0,Y 509.915,Z 330.596,A -85,B 0,C 180,E1 -5606.378,E2 -5606.378} C_VEL
LIN {X 0,Y 509.877,Z 330.594,A -85,B 0,C 180,E1 -5608.844,E2 -5608.844} C_VEL
LIN {X 0,Y 509.825,Z 330.601,A -85,B 0,C 180,E1 -5611.59,E2 -5611.59} C_VEL
LIN {X 0,Y 509.852,Z 330.6,A -85,B 0,C 180,E1 -5614.414,E2 -5614.414} C_VEL
LIN {X 0,Y 509.813,Z 330.603,A -85,B 0,C 180,E1 -5617.341,E2 -5617.341} C_VEL
LIN {X 0,Y 509.846,Z 330.599,A -85,B 0,C 180,E1 -5618.422,E2 -5618.422} C_VEL
LIN {X 0,Y 509.142,Z 330.685,A -85,B 0,C 180,E1 -5619.081,E2 -5619.081} C_VEL
LIN {X 0,Y 506.256,Z 331.048,A -85,B 0,C 180,E1 -5620.15,E2 -5620.15} C_VEL
LIN {X 0,Y 503.854,Z 331.344,A -85,B 0,C 180,E1 -5621.011,E2 -5621.011} C_VEL
LIN {X 0,Y 502.85,Z 331.475,A -85,B 0,C 180,E1 -5621.677,E2 -5621.677} C_VEL
LIN {X 0,Y 502.781,Z 331.479,A -85,B 0,C 180,E1 -5621.902,E2 -5621.902} C_VEL
LIN {X 0,Y 502.791,Z 331.477,A -85,B 0,C 180,E1 -5624.53,E2 -5624.53} C_VEL
LIN {X 0,Y 502.8,Z 331.481,A -85,B 0,C 180,E1 -5627.86,E2 -5627.86} C_VEL
LIN {X 0,Y 502.788,Z 331.479,A -85,B 0,C 180,E1 -5631.022,E2 -5631.022} C_VEL
LIN {X 0,Y 502.773,Z 331.48,A -85,B 0,C 180,E1 -5634.17,E2 -5634.17} C_VEL
LIN {X 0,Y 502.774,Z 331.483,A -85,B 0,C 180,E1 -5637.004,E2 -5637.004} C_VEL
LIN {X 0,Y 502.794,Z 331.479,A -85,B 0,C 180,E1 -5640.07,E2 -5640.07} C_VEL
LIN {X 0,Y 502.773,Z 331.481,A -85,B 0,C 180,E1 -5642.529,E2 -5642.529} C_VEL
LIN {X 0,Y 502.778,Z 331.505,A -85,B 0,C 180,E1 -5645.524,E2 -5645.524} C_VEL
LIN {X 0,Y 504.83,Z 342.342,A -85,B 0,C 180,E1 -5647.489,E2 -5647.489} C_VEL
LIN {X 0,Y 504.289,Z 357.585,A -85,B 0,C 180,E1 -5650.034,E2 -5650.034} C_VEL
LIN {X 0,Y 504.11,Z 362.774,A -85,B 0,C 180,E1 -5650.891,E2 -5650.891} C_VEL
LIN {X 0,Y 506.966,Z 377.944,A -85,B 0,C 180,E1 -5651.233,E2 -5651.233} C_VEL
LIN {X 0,Y 506.099,Z 499.372,A -85,B 0,C 180,E1 -5652.992,E2 -5652.992} C_VEL
LIN {X 0,Y 505.801,Z 513.995,A -85,B 0,C 180,E1 -5653.365,E2 -5653.365} C_VEL
LIN {X 0,Y 505.454,Z 528.233,A -85,B 0,C 180,E1 -5653.905,E2 -5653.905} C_VEL
LIN {X 0,Y 505.057,Z 541.242,A -85,B 0,C 180,E1 -5654.565,E2 -5654.565} C_VEL
LIN {X 0,Y 504.514,Z 553.839,A -85,B 0,C 180,E1 -5655.374,E2 -5655.374} C_VEL
LIN {X 0,Y 504.069,Z 565.318,A -85,B 0,C 180,E1 -5656.288,E2 -5656.288} C_VEL
LIN {X 0,Y 503.575,Z 576.042,A -85,B 0,C 180,E1 -5657.322,E2 -5657.322} C_VEL
LIN {X 0,Y 503.227,Z 586.298,A -85,B 0,C 180,E1 -5658.52,E2 -5658.52} C_VEL
LIN {X 0,Y 502.814,Z 594.92,A -85,B 0,C 180,E1 -5659.733,E2 -5659.733} C_VEL
LIN {X 0,Y 502.54,Z 603.185,A -85,B 0,C 180,E1 -5661.15,E2 -5661.15} C_VEL
LIN {X 0,Y 502.354,Z 608.944,A -85,B 0,C 180,E1 -5662.361,E2 -5662.361} C_VEL
LIN {X 0,Y 502.236,Z 613.682,A -85,B 0,C 180,E1 -5663.571,E2 -5663.571} C_VEL
LIN {X 0,Y 502.174,Z 617.525,A -85,B 0,C 180,E1 -5664.78,E2 -5664.78} C_VEL
LIN {X 0,Y 502.146,Z 620.472,A -85,B 0,C 180,E1 -5665.986,E2 -5665.986} C_VEL
LIN {X 0,Y 502.09,Z 623.189,A -85,B 0,C 180,E1 -5667.592,E2 -5667.592} C_VEL
LIN {X 0,Y 501.987,Z 624.558,A -85,B 0,C 180,E1 -5669.197,E2 -5669.197} C_VEL
LIN {X 0,Y 501.988,Z 624.602,A -85,B 0,C 180,E1 -5670.801,E2 -5670.801} C_VEL
LIN {X 0,Y 502.089,Z 623.32,A -85,B 0,C 180,E1 -5672.405,E2 -5672.405} C_VEL
LIN {X 0,Y 502.146,Z 620.681,A -85,B 0,C 180,E1 -5674.012,E2 -5674.012} C_VEL
LIN {X 0,Y 502.226,Z 616.612,A -85,B 0,C 180,E1 -5675.62,E2 -5675.62} C_VEL
LIN {X 0,Y 502.306,Z 610.993,A -85,B 0,C 180,E1 -5677.233,E2 -5677.233} C_VEL
LIN {X 0,Y 502.516,Z 604.654,A -85,B 0,C 180,E1 -5678.646,E2 -5678.646} C_VEL
LIN {X 0,Y 502.762,Z 596.768,A -85,B 0,C 180,E1 -5680.062,E2 -5680.062} C_VEL
LIN {X 0,Y 503.117,Z 588.518,A -85,B 0,C 180,E1 -5681.276,E2 -5681.276} C_VEL
LIN {X 0,Y 503.493,Z 578.583,A -85,B 0,C 180,E1 -5682.493,E2 -5682.493} C_VEL
LIN {X 0,Y 503.957,Z 567.518,A -85,B 0,C 180,E1 -5683.61,E2 -5683.61} C_VEL
LIN {X 0,Y 504.415,Z 556.51,A -85,B 0,C 180,E1 -5684.523,E2 -5684.523} C_VEL
LIN {X 0,Y 504.893,Z 544.565,A -85,B 0,C 180,E1 -5685.334,E2 -5685.334} C_VEL
LIN {X 0,Y 505.378,Z 531.366,A -85,B 0,C 180,E1 -5686.043,E2 -5686.043} C_VEL
LIN {X 0,Y 505.753,Z 517.128,A -85,B 0,C 180,E1 -5686.62,E2 -5686.62} C_VEL
LIN {X 0,Y 506.06,Z 502.334,A -85,B 0,C 180,E1 -5687.033,E2 -5687.033} C_VEL
LIN {X 0,Y 506.291,Z 480.13,A -85,B 0,C 180,E1 -5687.389,E2 -5687.389} C_VEL
LIN {X 0,Y 506.916,Z 376.99,A -85,B 0,C 180,E1 -5688.873,E2 -5688.873} C_VEL
LIN {X 0,Y 504.122,Z 362.664,A -85,B 0,C 180,E1 -5689.217,E2 -5689.217} C_VEL
LIN {X 0,Y 504.837,Z 344.158,A -85,B 0,C 180,E1 -5692.292,E2 -5692.292} C_VEL
LIN {X 0,Y 504.406,Z 339.345,A -85,B 0,C 180,E1 -5693.133,E2 -5693.133} C_VEL
LIN {X 0,Y 502.784,Z 331.485,A -85,B 0,C 180,E1 -5694.601,E2 -5694.601} C_VEL
LIN {X 0,Y 502.768,Z 331.485,A -85,B 0,C 180,E1 -5697.469,E2 -5697.469} C_VEL
LIN {X 0,Y 502.782,Z 331.48,A -85,B 0,C 180,E1 -5700.211,E2 -5700.211} C_VEL
LIN {X 0,Y 502.823,Z 331.481,A -85,B 0,C 180,E1 -5703.03,E2 -5703.03} C_VEL
LIN {X 0,Y 502.76,Z 331.481,A -85,B 0,C 180,E1 -5705.95,E2 -5705.95} C_VEL
LIN {X 0,Y 502.776,Z 331.485,A -85,B 0,C 180,E1 -5708.976,E2 -5708.976} C_VEL
LIN {X 0,Y 502.735,Z 331.484,A -85,B 0,C 180,E1 -5712.19,E2 -5712.19} C_VEL
LIN {X 0,Y 502.776,Z 331.479,A -85,B 0,C 180,E1 -5715.469,E2 -5715.469} C_VEL
LIN {X 0,Y 502.76,Z 331.487,A -85,B 0,C 180,E1 -5718.928,E2 -5718.928} C_VEL
LIN {X 0,Y 502.777,Z 331.474,A -85,B 0,C 180,E1 -5722.044,E2 -5722.044} C_VEL
LIN {X 0,Y 502.778,Z 331.482,A -85,B 0,C 180,E1 -5725.032,E2 -5725.032} C_VEL
LIN {X 0,Y 502.765,Z 331.474,A -85,B 0,C 180,E1 -5727.914,E2 -5727.914} C_VEL
LIN {X 0,Y 502.79,Z 331.484,A -85,B 0,C 180,E1 -5730.71,E2 -5730.71} C_VEL
LIN {X 0,Y 502.76,Z 331.472,A -85,B 0,C 180,E1 -5733.459,E2 -5733.459} C_VEL
LIN {X 0,Y 502.752,Z 331.48,A -85,B 0,C 180,E1 -5736.084,E2 -5736.084} C_VEL
LIN {X 0,Y 502.764,Z 331.483,A -85,B 0,C 180,E1 -5738.688,E2 -5738.688} C_VEL
LIN {X 0,Y 502.805,Z 331.469,A -85,B 0,C 180,E1 -5741.247,E2 -5741.247} C_VEL
LIN {X 0,Y 502.82,Z 331.481,A -85,B 0,C 180,E1 -5744.664,E2 -5744.664} C_VEL
LIN {X 0,Y 502.861,Z 331.467,A -85,B 0,C 180,E1 -5748.039,E2 -5748.039} C_VEL
LIN {X 0,Y 502.842,Z 331.47,A -85,B 0,C 180,E1 -5751.156,E2 -5751.156} C_VEL
LIN {X 0,Y 502.832,Z 331.47,A -85,B 0,C 180,E1 -5753.58,E2 -5753.58} C_VEL
LIN {X 0,Y 502.849,Z 331.474,A -85,B 0,C 180,E1 -5756.795,E2 -5756.795} C_VEL
LIN {X 0,Y 502.885,Z 331.47,A -85,B 0,C 180,E1 -5758.398,E2 -5758.398} C_VEL
LIN {X 0,Y 502.994,Z 331.456,A -85,B 0,C 180,E1 -5760.801,E2 -5760.801} C_VEL
LIN {X 0,Y 502.995,Z 331.457,A -85,B 0,C 180,E1 -5762.402,E2 -5762.402} C_VEL
LIN {X 0,Y 502.898,Z 331.462,A -85,B 0,C 180,E1 -5765.614,E2 -5765.614} C_VEL
LIN {X 0,Y 502.831,Z 331.473,A -85,B 0,C 180,E1 -5768.034,E2 -5768.034} C_VEL
LIN {X 0,Y 502.82,Z 331.472,A -85,B 0,C 180,E1 -5771.284,E2 -5771.284} C_VEL
LIN {X 0,Y 502.826,Z 331.478,A -85,B 0,C 180,E1 -5774.571,E2 -5774.571} C_VEL
LIN {X 0,Y 502.786,Z 331.477,A -85,B 0,C 180,E1 -5777.91,E2 -5777.91} C_VEL
LIN {X 0,Y 502.815,Z 331.475,A -85,B 0,C 180,E1 -5780.537,E2 -5780.537} C_VEL
LIN {X 0,Y 502.771,Z 331.475,A -85,B 0,C 180,E1 -5783.042,E2 -5783.042} C_VEL
LIN {X 0,Y 502.755,Z 331.481,A -85,B 0,C 180,E1 -5785.68,E2 -5785.68} C_VEL
LIN {X 0,Y 502.763,Z 331.48,A -85,B 0,C 180,E1 -5788.377,E2 -5788.377} C_VEL
LIN {X 0,Y 502.771,Z 331.478,A -85,B 0,C 180,E1 -5791.145,E2 -5791.145} C_VEL
LIN {X 0,Y 502.771,Z 331.481,A -85,B 0,C 180,E1 -5793.996,E2 -5793.996} C_VEL
LIN {X 0,Y 502.719,Z 331.485,A -85,B 0,C 180,E1 -5797.172,E2 -5797.172} C_VEL
LIN {X 0,Y 502.722,Z 331.49,A -85,B 0,C 180,E1 -5800.022,E2 -5800.022} C_VEL
LIN {X 0,Y 502.728,Z 331.483,A -85,B 0,C 180,E1 -5803.236,E2 -5803.236} C_VEL
LIN {X 0,Y 502.755,Z 331.482,A -85,B 0,C 180,E1 -5805.66,E2 -5805.66} C_VEL
LIN {X 0,Y 502.739,Z 331.484,A -85,B 0,C 180,E1 -5809.016,E2 -5809.016} C_VEL
LIN {X 0,Y 502.745,Z 331.489,A -85,B 0,C 180,E1 -5812.044,E2 -5812.044} C_VEL
LIN {X 0,Y 502.773,Z 331.48,A -85,B 0,C 180,E1 -5815.034,E2 -5815.034} C_VEL
LIN {X 0,Y 502.756,Z 331.487,A -85,B 0,C 180,E1 -5817.915,E2 -5817.915} C_VEL
LIN {X 0,Y 502.795,Z 331.476,A -85,B 0,C 180,E1 -5820.712,E2 -5820.712} C_VEL
LIN {X 0,Y 502.764,Z 331.483,A -85,B 0,C 180,E1 -5823.462,E2 -5823.462} C_VEL
LIN {X 0,Y 502.793,Z 331.679,A -85,B 0,C 180,E1 -5824.383,E2 -5824.383} C_VEL
LIN {X 0,Y 505.017,Z 342.111,A -85,B 0,C 180,E1 -5826.2,E2 -5826.2} C_VEL
LIN {X 0,Y 504.828,Z 351.535,A -85,B 0,C 180,E1 -5827.707,E2 -5827.707} C_VEL
LIN {X 0,Y 504.126,Z 371.364,A -85,B 0,C 180,E1 -5830.824,E2 -5830.824} C_VEL
LIN {X 0,Y 506.979,Z 387.475,A -85,B 0,C 180,E1 -5831.195,E2 -5831.195} C_VEL
LIN {X 0,Y 506.072,Z 509.533,A -85,B 0,C 180,E1 -5832.968,E2 -5832.968} C_VEL
LIN {X 0,Y 505.76,Z 523.975,A -85,B 0,C 180,E1 -5833.346,E2 -5833.346} C_VEL
LIN {X 0,Y 505.383,Z 537.327,A -85,B 0,C 180,E1 -5833.853,E2 -5833.853} C_VEL
LIN {X 0,Y 504.953,Z 551.276,A -85,B 0,C 180,E1 -5834.564,E2 -5834.564} C_VEL
LIN {X 0,Y 504.432,Z 563.747,A -85,B 0,C 180,E1 -5835.374,E2 -5835.374} C_VEL
LIN {X 0,Y 503.918,Z 576.309,A -85,B 0,C 180,E1 -5836.389,E2 -5836.389} C_VEL
LIN {X 0,Y 503.456,Z 587.506,A -85,B 0,C 180,E1 -5837.506,E2 -5837.506} C_VEL
LIN {X 0,Y 503.079,Z 597.54,A -85,B 0,C 180,E1 -5838.723,E2 -5838.723} C_VEL
LIN {X 0,Y 502.709,Z 605.875,A -85,B 0,C 180,E1 -5839.937,E2 -5839.937} C_VEL
LIN {X 0,Y 502.472,Z 613.844,A -85,B 0,C 180,E1 -5841.354,E2 -5841.354} C_VEL
LIN {X 0,Y 502.252,Z 620.256,A -85,B 0,C 180,E1 -5842.766,E2 -5842.766} C_VEL
LIN {X 0,Y 502.217,Z 625.945,A -85,B 0,C 180,E1 -5844.38,E2 -5844.38} C_VEL
LIN {X 0,Y 502.113,Z 630.072,A -85,B 0,C 180,E1 -5845.988,E2 -5845.988} C_VEL
LIN {X 0,Y 502.063,Z 632.764,A -85,B 0,C 180,E1 -5847.594,E2 -5847.594} C_VEL
LIN {X 0,Y 501.988,Z 634.095,A -85,B 0,C 180,E1 -5849.199,E2 -5849.199} C_VEL
LIN {X 0,Y 501.988,Z 634.093,A -85,B 0,C 180,E1 -5850.803,E2 -5850.803} C_VEL
LIN {X 0,Y 502.063,Z 632.758,A -85,B 0,C 180,E1 -5852.408,E2 -5852.408} C_VEL
LIN {X 0,Y 502.113,Z 630.063,A -85,B 0,C 180,E1 -5854.014,E2 -5854.014} C_VEL
LIN {X 0,Y 502.213,Z 625.937,A -85,B 0,C 180,E1 -5855.623,E2 -5855.623} C_VEL
LIN {X 0,Y 502.254,Z 620.248,A -85,B 0,C 180,E1 -5857.236,E2 -5857.236} C_VEL
LIN {X 0,Y 502.474,Z 613.831,A -85,B 0,C 180,E1 -5858.649,E2 -5858.649} C_VEL
LIN {X 0,Y 502.715,Z 605.861,A -85,B 0,C 180,E1 -5860.065,E2 -5860.065} C_VEL
LIN {X 0,Y 503.106,Z 597.523,A -85,B 0,C 180,E1 -5861.279,E2 -5861.279} C_VEL
LIN {X 0,Y 503.498,Z 586.845,A -85,B 0,C 180,E1 -5862.568,E2 -5862.568} C_VEL
LIN {X 0,Y 503.926,Z 576.283,A -85,B 0,C 180,E1 -5863.613,E2 -5863.613} C_VEL
LIN {X 0,Y 504.416,Z 565.136,A -85,B 0,C 180,E1 -5864.525,E2 -5864.525} C_VEL
LIN {X 0,Y 504.875,Z 553,A -85,B 0,C 180,E1 -5865.337,E2 -5865.337} C_VEL
LIN {X 0,Y 505.385,Z 539.545,A -85,B 0,C 180,E1 -5866.046,E2 -5866.046} C_VEL
LIN {X 0,Y 505.732,Z 525.159,A -85,B 0,C 180,E1 -5866.615,E2 -5866.615} C_VEL
LIN {X 0,Y 506.071,Z 510.567,A -85,B 0,C 180,E1 -5867.009,E2 -5867.009} C_VEL
LIN {X 0,Y 506.332,Z 484.235,A -85,B 0,C 180,E1 -5867.416,E2 -5867.416} C_VEL
LIN {X 0,Y 506.889,Z 386.215,A -85,B 0,C 180,E1 -5868.827,E2 -5868.827} C_VEL
LIN {X 0,Y 504.127,Z 371.416,A -85,B 0,C 180,E1 -5869.167,E2 -5869.167} C_VEL
LIN {X 0,Y 504.715,Z 354.209,A -85,B 0,C 180,E1 -5871.87,E2 -5871.87} C_VEL
LIN {X 0,Y 505.139,Z 344.009,A -85,B 0,C 180,E1 -5873.487,E2 -5873.487} C_VEL
LIN {X 0,Y 503.906,Z 336.693,A -85,B 0,C 180,E1 -5874.735,E2 -5874.735} C_VEL
LIN {X 0,Y 502.793,Z 331.483,A -85,B 0,C 180,E1 -5875.679,E2 -5875.679} C_VEL
LIN {X 0,Y 502.773,Z 331.481,A -85,B 0,C 180,E1 -5878.378,E2 -5878.378} C_VEL
LIN {X 0,Y 502.796,Z 331.482,A -85,B 0,C 180,E1 -5881.144,E2 -5881.144} C_VEL
LIN {X 0,Y 502.807,Z 331.476,A -85,B 0,C 180,E1 -5883.995,E2 -5883.995} C_VEL
LIN {X 0,Y 502.77,Z 331.485,A -85,B 0,C 180,E1 -5887.176,E2 -5887.176} C_VEL
LIN {X 0,Y 502.793,Z 331.476,A -85,B 0,C 180,E1 -5890.016,E2 -5890.016} C_VEL
LIN {X 0,Y 502.808,Z 331.475,A -85,B 0,C 180,E1 -5892.2,E2 -5892.2} C_VEL
LIN {X 0,Y 502.806,Z 331.476,A -85,B 0,C 180,E1 -5895.469,E2 -5895.469} C_VEL
LIN {X 0,Y 502.825,Z 331.477,A -85,B 0,C 180,E1 -5898.935,E2 -5898.935} C_VEL
LIN {X 0,Y 502.795,Z 331.479,A -85,B 0,C 180,E1 -5902.046,E2 -5902.046} C_VEL
LIN {X 0,Y 502.802,Z 331.477,A -85,B 0,C 180,E1 -5905.034,E2 -5905.034} C_VEL
LIN {X 0,Y 502.788,Z 331.483,A -85,B 0,C 180,E1 -5907.916,E2 -5907.916} C_VEL
LIN {X 0,Y 502.817,Z 331.48,A -85,B 0,C 180,E1 -5910.712,E2 -5910.712} C_VEL
LIN {X 0,Y 502.778,Z 331.485,A -85,B 0,C 180,E1 -5913.46,E2 -5913.46} C_VEL
LIN {X 0,Y 502.774,Z 331.487,A -85,B 0,C 180,E1 -5916.085,E2 -5916.085} C_VEL
LIN {X 0,Y 502.875,Z 331.637,A -85,B 0,C 180,E1 -5917.143,E2 -5917.143} C_VEL
LIN {X 0,Y 504.068,Z 338.636,A -85,B 0,C 180,E1 -5918.317,E2 -5918.317} C_VEL
LIN {X 0,Y 503.893,Z 355.66,A -85,B 0,C 180,E1 -5921.078,E2 -5921.078} C_VEL
LIN {X 0,Y 503.63,Z 373.409,A -85,B 0,C 180,E1 -5923.977,E2 -5923.977} C_VEL
LIN {X 0,Y 503.591,Z 375.294,A -85,B 0,C 180,E1 -5924.286,E2 -5924.286} C_VEL
LIN {X 0,Y 505.366,Z 386.277,A -85,B 0,C 180,E1 -5924.529,E2 -5924.529} C_VEL
LIN {X 0,Y 504.637,Z 483.604,A -85,B 0,C 180,E1 -5926.048,E2 -5926.048} C_VEL
LIN {X 0,Y 504.417,Z 496.586,A -85,B 0,C 180,E1 -5926.401,E2 -5926.401} C_VEL
LIN {X 0,Y 504.154,Z 509.003,A -85,B 0,C 180,E1 -5926.907,E2 -5926.907} C_VEL
LIN {X 0,Y 503.892,Z 521.164,A -85,B 0,C 180,E1 -5927.572,E2 -5927.572} C_VEL
LIN {X 0,Y 503.642,Z 531.886,A -85,B 0,C 180,E1 -5928.326,E2 -5928.326} C_VEL
LIN {X 0,Y 503.249,Z 543.294,A -85,B 0,C 180,E1 -5929.337,E2 -5929.337} C_VEL
LIN {X 0,Y 502.938,Z 552.471,A -85,B 0,C 180,E1 -5930.347,E2 -5930.347} C_VEL
LIN {X 0,Y 502.664,Z 561.293,A -85,B 0,C 180,E1 -5931.558,E2 -5931.558} C_VEL
LIN {X 0,Y 502.482,Z 568.395,A -85,B 0,C 180,E1 -5932.769,E2 -5932.769} C_VEL
LIN {X 0,Y 502.373,Z 574.05,A -85,B 0,C 180,E1 -5933.977,E2 -5933.977} C_VEL
LIN {X 0,Y 502.145,Z 578.464,A -85,B 0,C 180,E1 -5935.183,E2 -5935.183} C_VEL
LIN {X 0,Y 502.239,Z 580.766,A -85,B 0,C 180,E1 -5935.988,E2 -5935.988} C_VEL
LIN {X 0,Y 502.18,Z 582.65,A -85,B 0,C 180,E1 -5936.791,E2 -5936.791} C_VEL
LIN {X 0,Y 502.128,Z 584.105,A -85,B 0,C 180,E1 -5937.594,E2 -5937.594} C_VEL
LIN {X 0,Y 501.994,Z 585.732,A -85,B 0,C 180,E1 -5939.198,E2 -5939.198} C_VEL
LIN {X 0,Y 501.987,Z 585.965,A -85,B 0,C 180,E1 -5940,E2 -5940} C_VEL
LIN {X 0,Y 501.994,Z 585.765,A -85,B 0,C 180,E1 -5940.802,E2 -5940.802} C_VEL
LIN {X 0,Y 502.124,Z 584.166,A -85,B 0,C 180,E1 -5942.407,E2 -5942.407} C_VEL
LIN {X 0,Y 502.147,Z 582.768,A -85,B 0,C 180,E1 -5943.209,E2 -5943.209} C_VEL
LIN {X 0,Y 502.216,Z 579.84,A -85,B 0,C 180,E1 -5944.414,E2 -5944.414} C_VEL
LIN {X 0,Y 502.294,Z 575.861,A -85,B 0,C 180,E1 -5945.621,E2 -5945.621} C_VEL
LIN {X 0,Y 502.383,Z 570.121,A -85,B 0,C 180,E1 -5946.95,E2 -5946.95} C_VEL
LIN {X 0,Y 502.609,Z 563.024,A -85,B 0,C 180,E1 -5948.24,E2 -5948.24} C_VEL
LIN {X 0,Y 502.856,Z 554.629,A -85,B 0,C 180,E1 -5949.452,E2 -5949.452} C_VEL
LIN {X 0,Y 503.091,Z 546.011,A -85,B 0,C 180,E1 -5950.463,E2 -5950.463} C_VEL
LIN {X 0,Y 503.495,Z 535.437,A -85,B 0,C 180,E1 -5951.473,E2 -5951.473} C_VEL
LIN {X 0,Y 503.775,Z 524.36,A -85,B 0,C 180,E1 -5952.314,E2 -5952.314} C_VEL
LIN {X 0,Y 504.115,Z 513.066,A -85,B 0,C 180,E1 -5952.991,E2 -5952.991} C_VEL
LIN {X 0,Y 504.402,Z 500.963,A -85,B 0,C 180,E1 -5953.548,E2 -5953.548} C_VEL
LIN {X 0,Y 504.604,Z 488.488,A -85,B 0,C 180,E1 -5953.953,E2 -5953.953} C_VEL
LIN {X 0,Y 504.764,Z 474.593,A -85,B 0,C 180,E1 -5954.231,E2 -5954.231} C_VEL
LIN {X 0,Y 505.302,Z 384.898,A -85,B 0,C 180,E1 -5955.592,E2 -5955.592} C_VEL
LIN {X 0,Y 503.476,Z 374.499,A -85,B 0,C 180,E1 -5955.813,E2 -5955.813} C_VEL
LIN {X 0,Y 503.879,Z 356.013,A -85,B 0,C 180,E1 -5958.922,E2 -5958.922} C_VEL
LIN {X 0,Y 504.142,Z 339.727,A -85,B 0,C 180,E1 -5961.68,E2 -5961.68} C_VEL
LIN {X 0,Y 502.822,Z 331.477,A -85,B 0,C 180,E1 -5963.148,E2 -5963.148} C_VEL
LIN {X 0,Y 502.87,Z 331.471,A -85,B 0,C 180,E1 -5966.566,E2 -5966.566} C_VEL
LIN {X 0,Y 502.828,Z 331.472,A -85,B 0,C 180,E1 -5969.288,E2 -5969.288} C_VEL
LIN {X 0,Y 502.789,Z 331.484,A -85,B 0,C 180,E1 -5972.084,E2 -5972.084} C_VEL
LIN {X 0,Y 502.803,Z 331.475,A -85,B 0,C 180,E1 -5974.966,E2 -5974.966} C_VEL
LIN {X 0,Y 502.796,Z 331.477,A -85,B 0,C 180,E1 -5978.485,E2 -5978.485} C_VEL
LIN {X 0,Y 502.783,Z 331.477,A -85,B 0,C 180,E1 -5981.07,E2 -5981.07} C_VEL
LIN {X 0,Y 502.781,Z 331.479,A -85,B 0,C 180,E1 -5981.902,E2 -5981.902} C_VEL
LIN {X 0,Y 502.15,Z 331.562,A -85,B 0,C 180,E1 -5982.57,E2 -5982.57} C_VEL
LIN {X 0,Y 499.304,Z 331.917,A -85,B 0,C 180,E1 -5983.656,E2 -5983.656} C_VEL
LIN {X 0,Y 496.87,Z 332.217,A -85,B 0,C 180,E1 -5984.53,E2 -5984.53} C_VEL
LIN {X 0,Y 495.815,Z 332.348,A -85,B 0,C 180,E1 -5985.206,E2 -5985.206} C_VEL
LIN {X 0,Y 495.725,Z 332.358,A -85,B 0,C 180,E1 -5985.435,E2 -5985.435} C_VEL
LIN {X 0,Y 495.722,Z 332.357,A -85,B 0,C 180,E1 -5988.712,E2 -5988.712} C_VEL
LIN {X 0,Y 495.729,Z 332.363,A -85,B 0,C 180,E1 -5991.405,E2 -5991.405} C_VEL
LIN {X 0,Y 495.746,Z 332.354,A -85,B 0,C 180,E1 -5994.461,E2 -5994.461} C_VEL
LIN {X 0,Y 495.729,Z 332.361,A -85,B 0,C 180,E1 -5997.402,E2 -5997.402} C_VEL
LIN {X 0,Y 495.743,Z 332.357,A -85,B 0,C 180,E1 -6000.251,E2 -6000.251} C_VEL
LIN {X 0,Y 495.724,Z 332.359,A -85,B 0,C 180,E1 -6003.274,E2 -6003.274} C_VEL
LIN {X 0,Y 495.735,Z 332.417,A -85,B 0,C 180,E1 -6005.303,E2 -6005.303} C_VEL
LIN {X 0,Y 497.927,Z 343.673,A -85,B 0,C 180,E1 -6007.379,E2 -6007.379} C_VEL
LIN {X 0,Y 497.407,Z 357.652,A -85,B 0,C 180,E1 -6009.746,E2 -6009.746} C_VEL
LIN {X 0,Y 497.209,Z 362.875,A -85,B 0,C 180,E1 -6010.62,E2 -6010.62} C_VEL
LIN {X 0,Y 500.233,Z 378.054,A -85,B 0,C 180,E1 -6010.971,E2 -6010.971} C_VEL
LIN {X 0,Y 499.326,Z 499.473,A -85,B 0,C 180,E1 -6012.754,E2 -6012.754} C_VEL
LIN {X 0,Y 499.009,Z 513.862,A -85,B 0,C 180,E1 -6013.124,E2 -6013.124} C_VEL
LIN {X 0,Y 498.69,Z 527.186,A -85,B 0,C 180,E1 -6013.628,E2 -6013.628} C_VEL
LIN {X 0,Y 498.269,Z 539.558,A -85,B 0,C 180,E1 -6014.244,E2 -6014.244} C_VEL
LIN {X 0,Y 497.717,Z 552.492,A -85,B 0,C 180,E1 -6015.065,E2 -6015.065} C_VEL
LIN {X 0,Y 497.18,Z 564.221,A -85,B 0,C 180,E1 -6015.99,E2 -6015.99} C_VEL
LIN {X 0,Y 496.681,Z 575.045,A -85,B 0,C 180,E1 -6017.028,E2 -6017.028} C_VEL
LIN {X 0,Y 496.318,Z 584.911,A -85,B 0,C 180,E1 -6018.171,E2 -6018.171} C_VEL
LIN {X 0,Y 495.849,Z 593.641,A -85,B 0,C 180,E1 -6019.381,E2 -6019.381} C_VEL
LIN {X 0,Y 495.554,Z 602.153,A -85,B 0,C 180,E1 -6020.818,E2 -6020.818} C_VEL
LIN {X 0,Y 495.294,Z 609.015,A -85,B 0,C 180,E1 -6022.252,E2 -6022.252} C_VEL
LIN {X 0,Y 495.146,Z 614.676,A -85,B 0,C 180,E1 -6023.745,E2 -6023.745} C_VEL
LIN {X 0,Y 495.032,Z 618.655,A -85,B 0,C 180,E1 -6025.112,E2 -6025.112} C_VEL
LIN {X 0,Y 495.038,Z 622.071,A -85,B 0,C 180,E1 -6026.743,E2 -6026.743} C_VEL
LIN {X 0,Y 494.961,Z 624.107,A -85,B 0,C 180,E1 -6028.371,E2 -6028.371} C_VEL
LIN {X 0,Y 494.897,Z 624.813,A -85,B 0,C 180,E1 -6029.999,E2 -6029.999} C_VEL
LIN {X 0,Y 494.96,Z 624.194,A -85,B 0,C 180,E1 -6031.626,E2 -6031.626} C_VEL
LIN {X 0,Y 495.037,Z 622.239,A -85,B 0,C 180,E1 -6033.254,E2 -6033.254} C_VEL
LIN {X 0,Y 495.031,Z 618.898,A -85,B 0,C 180,E1 -6034.885,E2 -6034.885} C_VEL
LIN {X 0,Y 495.143,Z 614.996,A -85,B 0,C 180,E1 -6036.252,E2 -6036.252} C_VEL
LIN {X 0,Y 495.288,Z 609.42,A -85,B 0,C 180,E1 -6037.746,E2 -6037.746} C_VEL
LIN {X 0,Y 495.548,Z 602.654,A -85,B 0,C 180,E1 -6039.179,E2 -6039.179} C_VEL
LIN {X 0,Y 495.82,Z 594.246,A -85,B 0,C 180,E1 -6040.617,E2 -6040.617} C_VEL
LIN {X 0,Y 496.3,Z 584.531,A -85,B 0,C 180,E1 -6041.968,E2 -6041.968} C_VEL
LIN {X 0,Y 496.684,Z 574.839,A -85,B 0,C 180,E1 -6043.084,E2 -6043.084} C_VEL
LIN {X 0,Y 497.211,Z 564.088,A -85,B 0,C 180,E1 -6044.111,E2 -6044.111} C_VEL
LIN {X 0,Y 497.718,Z 552.33,A -85,B 0,C 180,E1 -6045.037,E2 -6045.037} C_VEL
LIN {X 0,Y 498.27,Z 539.346,A -85,B 0,C 180,E1 -6045.858,E2 -6045.858} C_VEL
LIN {X 0,Y 498.745,Z 526.177,A -85,B 0,C 180,E1 -6046.507,E2 -6046.507} C_VEL
LIN {X 0,Y 499.095,Z 511.894,A -85,B 0,C 180,E1 -6047.025,E2 -6047.025} C_VEL
LIN {X 0,Y 499.349,Z 497.254,A -85,B 0,C 180,E1 -6047.374,E2 -6047.374} C_VEL
LIN {X 0,Y 500.3,Z 378.609,A -85,B 0,C 180,E1 -6049.109,E2 -6049.109} C_VEL
LIN {X 0,Y 497.218,Z 362.879,A -85,B 0,C 180,E1 -6049.469,E2 -6049.469} C_VEL
LIN {X 0,Y 497.93,Z 345.485,A -85,B 0,C 180,E1 -6052.4,E2 -6052.4} C_VEL
LIN {X 0,Y 497.558,Z 341.201,A -85,B 0,C 180,E1 -6053.158,E2 -6053.158} C_VEL
LIN {X 0,Y 495.716,Z 332.366,A -85,B 0,C 180,E1 -6054.827,E2 -6054.827} C_VEL
LIN {X 0,Y 495.709,Z 332.362,A -85,B 0,C 180,E1 -6057.894,E2 -6057.894} C_VEL
LIN {X 0,Y 495.732,Z 332.363,A -85,B 0,C 180,E1 -6060.687,E2 -6060.687} C_VEL
LIN {X 0,Y 495.744,Z 332.358,A -85,B 0,C 180,E1 -6063.564,E2 -6063.564} C_VEL
LIN {X 0,Y 495.708,Z 332.363,A -85,B 0,C 180,E1 -6066.544,E2 -6066.544} C_VEL
LIN {X 0,Y 495.733,Z 332.356,A -85,B 0,C 180,E1 -6069.638,E2 -6069.638} C_VEL
LIN {X 0,Y 495.685,Z 332.368,A -85,B 0,C 180,E1 -6072.885,E2 -6072.885} C_VEL
LIN {X 0,Y 495.713,Z 332.358,A -85,B 0,C 180,E1 -6075.996,E2 -6075.996} C_VEL
LIN {X 0,Y 495.72,Z 332.36,A -85,B 0,C 180,E1 -6079.295,E2 -6079.295} C_VEL
LIN {X 0,Y 495.734,Z 332.352,A -85,B 0,C 180,E1 -6081.407,E2 -6081.407} C_VEL
LIN {X 0,Y 495.73,Z 332.359,A -85,B 0,C 180,E1 -6084.461,E2 -6084.461} C_VEL
LIN {X 0,Y 495.737,Z 332.35,A -85,B 0,C 180,E1 -6087.403,E2 -6087.403} C_VEL
LIN {X 0,Y 495.743,Z 332.356,A -85,B 0,C 180,E1 -6090.252,E2 -6090.252} C_VEL
LIN {X 0,Y 495.725,Z 332.35,A -85,B 0,C 180,E1 -6093.27,E2 -6093.27} C_VEL
LIN {X 0,Y 495.724,Z 332.362,A -85,B 0,C 180,E1 -6096.611,E2 -6096.611} C_VEL
LIN {X 0,Y 495.764,Z 332.347,A -85,B 0,C 180,E1 -6099.323,E2 -6099.323} C_VEL
LIN {X 0,Y 495.764,Z 332.344,A -85,B 0,C 180,E1 -6101.828,E2 -6101.828} C_VEL
LIN {X 0,Y 495.759,Z 332.353,A -85,B 0,C 180,E1 -6105.216,E2 -6105.216} C_VEL
LIN {X 0,Y 495.833,Z 332.349,A -85,B 0,C 180,E1 -6108.554,E2 -6108.554} C_VEL
LIN {X 0,Y 495.813,Z 332.344,A -85,B 0,C 180,E1 -6111.851,E2 -6111.851} C_VEL
LIN {X 0,Y 495.797,Z 332.346,A -85,B 0,C 180,E1 -6115.121,E2 -6115.121} C_VEL
LIN {X 0,Y 495.964,Z 332.326,A -85,B 0,C 180,E1 -6117.563,E2 -6117.563} C_VEL
LIN {X 0,Y 495.945,Z 332.333,A -85,B 0,C 180,E1 -6120.812,E2 -6120.812} C_VEL
LIN {X 0,Y 495.963,Z 332.333,A -85,B 0,C 180,E1 -6122.436,E2 -6122.436} C_VEL
LIN {X 0,Y 495.853,Z 332.34,A -85,B 0,C 180,E1 -6125.694,E2 -6125.694} C_VEL
LIN {X 0,Y 495.795,Z 332.35,A -85,B 0,C 180,E1 -6128.149,E2 -6128.149} C_VEL
LIN {X 0,Y 495.805,Z 332.345,A -85,B 0,C 180,E1 -6131.446,E2 -6131.446} C_VEL
LIN {X 0,Y 495.772,Z 332.354,A -85,B 0,C 180,E1 -6134.783,E2 -6134.783} C_VEL
LIN {X 0,Y 495.764,Z 332.355,A -85,B 0,C 180,E1 -6138.172,E2 -6138.172} C_VEL
LIN {X 0,Y 495.76,Z 332.35,A -85,B 0,C 180,E1 -6140.757,E2 -6140.757} C_VEL
LIN {X 0,Y 495.723,Z 332.351,A -85,B 0,C 180,E1 -6143.388,E2 -6143.388} C_VEL
LIN {X 0,Y 495.723,Z 332.358,A -85,B 0,C 180,E1 -6146.73,E2 -6146.73} C_VEL
LIN {X 0,Y 495.744,Z 332.349,A -85,B 0,C 180,E1 -6149.748,E2 -6149.748} C_VEL
LIN {X 0,Y 495.736,Z 332.358,A -85,B 0,C 180,E1 -6152.597,E2 -6152.597} C_VEL
LIN {X 0,Y 495.714,Z 332.358,A -85,B 0,C 180,E1 -6155.54,E2 -6155.54} C_VEL
LIN {X 0,Y 495.722,Z 332.359,A -85,B 0,C 180,E1 -6158.765,E2 -6158.765} C_VEL
LIN {X 0,Y 495.69,Z 332.362,A -85,B 0,C 180,E1 -6161.788,E2 -6161.788} C_VEL
LIN {X 0,Y 495.72,Z 332.357,A -85,B 0,C 180,E1 -6165.143,E2 -6165.143} C_VEL
LIN {X 0,Y 495.689,Z 332.369,A -85,B 0,C 180,E1 -6168.214,E2 -6168.214} C_VEL
LIN {X 0,Y 495.704,Z 332.36,A -85,B 0,C 180,E1 -6171.406,E2 -6171.406} C_VEL
LIN {X 0,Y 495.719,Z 332.363,A -85,B 0,C 180,E1 -6174.462,E2 -6174.462} C_VEL
LIN {X 0,Y 495.735,Z 332.357,A -85,B 0,C 180,E1 -6177.405,E2 -6177.405} C_VEL
LIN {X 0,Y 495.749,Z 332.357,A -85,B 0,C 180,E1 -6180.254,E2 -6180.254} C_VEL
LIN {X 0,Y 495.715,Z 332.361,A -85,B 0,C 180,E1 -6183.276,E2 -6183.276} C_VEL
LIN {X 0,Y 495.751,Z 332.441,A -85,B 0,C 180,E1 -6184.129,E2 -6184.129} C_VEL
LIN {X 0,Y 498.184,Z 344.371,A -85,B 0,C 180,E1 -6186.233,E2 -6186.233} C_VEL
LIN {X 0,Y 497.596,Z 360.944,A -85,B 0,C 180,E1 -6188.899,E2 -6188.899} C_VEL
LIN {X 0,Y 497.242,Z 371.59,A -85,B 0,C 180,E1 -6190.575,E2 -6190.575} C_VEL
LIN {X 0,Y 500.247,Z 388.546,A -85,B 0,C 180,E1 -6190.949,E2 -6190.949} C_VEL
LIN {X 0,Y 499.29,Z 509.466,A -85,B 0,C 180,E1 -6192.729,E2 -6192.729} C_VEL
LIN {X 0,Y 498.934,Z 523.631,A -85,B 0,C 180,E1 -6193.102,E2 -6193.102} C_VEL
LIN {X 0,Y 498.574,Z 537.26,A -85,B 0,C 180,E1 -6193.626,E2 -6193.626} C_VEL
LIN {X 0,Y 498.17,Z 549.44,A -85,B 0,C 180,E1 -6194.244,E2 -6194.244} C_VEL
LIN {X 0,Y 497.631,Z 562.253,A -85,B 0,C 180,E1 -6195.065,E2 -6195.065} C_VEL
LIN {X 0,Y 497.122,Z 573.894,A -85,B 0,C 180,E1 -6195.991,E2 -6195.991} C_VEL
LIN {X 0,Y 496.562,Z 584.659,A -85,B 0,C 180,E1 -6197.028,E2 -6197.028} C_VEL
LIN {X 0,Y 496.207,Z 594.54,A -85,B 0,C 180,E1 -6198.178,E2 -6198.178} C_VEL
LIN {X 0,Y 495.827,Z 603.186,A -85,B 0,C 180,E1 -6199.383,E2 -6199.383} C_VEL
LIN {X 0,Y 495.478,Z 611.68,A -85,B 0,C 180,E1 -6200.819,E2 -6200.819} C_VEL
LIN {X 0,Y 495.237,Z 618.521,A -85,B 0,C 180,E1 -6202.253,E2 -6202.253} C_VEL
LIN {X 0,Y 495.131,Z 624.188,A -85,B 0,C 180,E1 -6203.754,E2 -6203.754} C_VEL
LIN {X 0,Y 495.031,Z 628.127,A -85,B 0,C 180,E1 -6205.115,E2 -6205.115} C_VEL
LIN {X 0,Y 495.033,Z 631.525,A -85,B 0,C 180,E1 -6206.746,E2 -6206.746} C_VEL
LIN {X 0,Y 494.958,Z 633.53,A -85,B 0,C 180,E1 -6208.374,E2 -6208.374} C_VEL
LIN {X 0,Y 494.896,Z 634.193,A -85,B 0,C 180,E1 -6210.001,E2 -6210.001} C_VEL
LIN {X 0,Y 494.958,Z 633.526,A -85,B 0,C 180,E1 -6211.629,E2 -6211.629} C_VEL
LIN {X 0,Y 495.033,Z 631.516,A -85,B 0,C 180,E1 -6213.257,E2 -6213.257} C_VEL
LIN {X 0,Y 495.031,Z 628.118,A -85,B 0,C 180,E1 -6214.888,E2 -6214.888} C_VEL
LIN {X 0,Y 495.129,Z 623.356,A -85,B 0,C 180,E1 -6216.485,E2 -6216.485} C_VEL
LIN {X 0,Y 495.239,Z 618.512,A -85,B 0,C 180,E1 -6217.749,E2 -6217.749} C_VEL
LIN {X 0,Y 495.48,Z 611.666,A -85,B 0,C 180,E1 -6219.183,E2 -6219.183} C_VEL
LIN {X 0,Y 495.83,Z 603.17,A -85,B 0,C 180,E1 -6220.619,E2 -6220.619} C_VEL
LIN {X 0,Y 496.205,Z 593.424,A -85,B 0,C 180,E1 -6221.964,E2 -6221.964} C_VEL
LIN {X 0,Y 496.645,Z 583.562,A -85,B 0,C 180,E1 -6223.087,E2 -6223.087} C_VEL
LIN {X 0,Y 497.156,Z 572.691,A -85,B 0,C 180,E1 -6224.115,E2 -6224.115} C_VEL
LIN {X 0,Y 497.663,Z 560.788,A -85,B 0,C 180,E1 -6225.041,E2 -6225.041} C_VEL
LIN {X 0,Y 498.208,Z 547.623,A -85,B 0,C 180,E1 -6225.863,E2 -6225.863} C_VEL
LIN {X 0,Y 498.698,Z 534.104,A -85,B 0,C 180,E1 -6226.512,E2 -6226.512} C_VEL
LIN {X 0,Y 499.028,Z 520.247,A -85,B 0,C 180,E1 -6227.003,E2 -6227.003} C_VEL
LIN {X 0,Y 499.353,Z 506.588,A -85,B 0,C 180,E1 -6227.324,E2 -6227.324} C_VEL
LIN {X 0,Y 500.199,Z 387.219,A -85,B 0,C 180,E1 -6229.073,E2 -6229.073} C_VEL
LIN {X 0,Y 497.205,Z 371.349,A -85,B 0,C 180,E1 -6229.445,E2 -6229.445} C_VEL
LIN {X 0,Y 497.883,Z 352.8,A -85,B 0,C 180,E1 -6232.404,E2 -6232.404} C_VEL
LIN {X 0,Y 498.174,Z 344.353,A -85,B 0,C 180,E1 -6233.769,E2 -6233.769} C_VEL
LIN {X 0,Y 495.738,Z 332.362,A -85,B 0,C 180,E1 -6235.902,E2 -6235.902} C_VEL
LIN {X 0,Y 495.728,Z 332.359,A -85,B 0,C 180,E1 -6238.819,E2 -6238.819} C_VEL
LIN {X 0,Y 495.758,Z 332.359,A -85,B 0,C 180,E1 -6241.726,E2 -6241.726} C_VEL
LIN {X 0,Y 495.772,Z 332.353,A -85,B 0,C 180,E1 -6244.694,E2 -6244.694} C_VEL
LIN {X 0,Y 495.726,Z 332.359,A -85,B 0,C 180,E1 -6247.563,E2 -6247.563} C_VEL
LIN {X 0,Y 495.764,Z 332.351,A -85,B 0,C 180,E1 -6250.048,E2 -6250.048} C_VEL
LIN {X 0,Y 495.73,Z 332.361,A -85,B 0,C 180,E1 -6252.884,E2 -6252.884} C_VEL
LIN {X 0,Y 495.739,Z 332.356,A -85,B 0,C 180,E1 -6256,E2 -6256} C_VEL
LIN {X 0,Y 495.771,Z 332.352,A -85,B 0,C 180,E1 -6259.301,E2 -6259.301} C_VEL
LIN {X 0,Y 495.726,Z 332.362,A -85,B 0,C 180,E1 -6262.438,E2 -6262.438} C_VEL
LIN {X 0,Y 495.782,Z 332.351,A -85,B 0,C 180,E1 -6265.457,E2 -6265.457} C_VEL
LIN {X 0,Y 495.76,Z 332.361,A -85,B 0,C 180,E1 -6268.364,E2 -6268.364} C_VEL
LIN {X 0,Y 495.758,Z 332.36,A -85,B 0,C 180,E1 -6271.515,E2 -6271.515} C_VEL
LIN {X 0,Y 495.721,Z 332.366,A -85,B 0,C 180,E1 -6273.928,E2 -6273.928} C_VEL
LIN {X 0,Y 495.814,Z 332.52,A -85,B 0,C 180,E1 -6276.955,E2 -6276.955} C_VEL
LIN {X 0,Y 497.156,Z 339.988,A -85,B 0,C 180,E1 -6278.218,E2 -6278.218} C_VEL
LIN {X 0,Y 497.01,Z 355.906,A -85,B 0,C 180,E1 -6280.806,E2 -6280.806} C_VEL
LIN {X 0,Y 496.7,Z 375.108,A -85,B 0,C 180,E1 -6283.966,E2 -6283.966} C_VEL
LIN {X 0,Y 496.684,Z 375.677,A -85,B 0,C 180,E1 -6284.06,E2 -6284.06} C_VEL
LIN {X 0,Y 498.553,Z 386.707,A -85,B 0,C 180,E1 -6284.313,E2 -6284.313} C_VEL
LIN {X 0,Y 497.72,Z 484.056,A -85,B 0,C 180,E1 -6285.876,E2 -6285.876} C_VEL
LIN {X 0,Y 497.535,Z 496.207,A -85,B 0,C 180,E1 -6286.21,E2 -6286.21} C_VEL
LIN {X 0,Y 497.219,Z 508.843,A -85,B 0,C 180,E1 -6286.721,E2 -6286.721} C_VEL
LIN {X 0,Y 496.951,Z 520.776,A -85,B 0,C 180,E1 -6287.375,E2 -6287.375} C_VEL
LIN {X 0,Y 496.684,Z 531.932,A -85,B 0,C 180,E1 -6288.16,E2 -6288.16} C_VEL
LIN {X 0,Y 496.316,Z 542.358,A -85,B 0,C 180,E1 -6289.083,E2 -6289.083} C_VEL
LIN {X 0,Y 495.94,Z 552.632,A -85,B 0,C 180,E1 -6290.209,E2 -6290.209} C_VEL
LIN {X 0,Y 495.626,Z 561.503,A -85,B 0,C 180,E1 -6291.437,E2 -6291.437} C_VEL
LIN {X 0,Y 495.427,Z 568.639,A -85,B 0,C 180,E1 -6292.665,E2 -6292.665} C_VEL
LIN {X 0,Y 495.316,Z 574.324,A -85,B 0,C 180,E1 -6293.891,E2 -6293.891} C_VEL
LIN {X 0,Y 495.068,Z 578.761,A -85,B 0,C 180,E1 -6295.114,E2 -6295.114} C_VEL
LIN {X 0,Y 495.175,Z 581.071,A -85,B 0,C 180,E1 -6295.931,E2 -6295.931} C_VEL
LIN {X 0,Y 495.101,Z 582.962,A -85,B 0,C 180,E1 -6296.745,E2 -6296.745} C_VEL
LIN {X 0,Y 495.063,Z 584.424,A -85,B 0,C 180,E1 -6297.559,E2 -6297.559} C_VEL
LIN {X 0,Y 494.914,Z 586.056,A -85,B 0,C 180,E1 -6299.186,E2 -6299.186} C_VEL
LIN {X 0,Y 494.904,Z 586.287,A -85,B 0,C 180,E1 -6300,E2 -6300} C_VEL
LIN {X 0,Y 494.914,Z 586.083,A -85,B 0,C 180,E1 -6300.814,E2 -6300.814} C_VEL
LIN {X 0,Y 495.058,Z 584.472,A -85,B 0,C 180,E1 -6302.441,E2 -6302.441} C_VEL
LIN {X 0,Y 495.071,Z 583.062,A -85,B 0,C 180,E1 -6303.255,E2 -6303.255} C_VEL
LIN {X 0,Y 495.143,Z 580.115,A -85,B 0,C 180,E1 -6304.478,E2 -6304.478} C_VEL
LIN {X 0,Y 495.242,Z 576.111,A -85,B 0,C 180,E1 -6305.701,E2 -6305.701} C_VEL
LIN {X 0,Y 495.335,Z 570.045,A -85,B 0,C 180,E1 -6307.111,E2 -6307.111} C_VEL
LIN {X 0,Y 495.571,Z 563.21,A -85,B 0,C 180,E1 -6308.358,E2 -6308.358} C_VEL
LIN {X 0,Y 495.829,Z 554.766,A -85,B 0,C 180,E1 -6309.587,E2 -6309.587} C_VEL
LIN {X 0,Y 496.098,Z 546.103,A -85,B 0,C 180,E1 -6310.613,E2 -6310.613} C_VEL
LIN {X 0,Y 496.522,Z 535.462,A -85,B 0,C 180,E1 -6311.637,E2 -6311.637} C_VEL
LIN {X 0,Y 496.837,Z 523.54,A -85,B 0,C 180,E1 -6312.542,E2 -6312.542} C_VEL
LIN {X 0,Y 497.182,Z 512.933,A -85,B 0,C 180,E1 -6313.176,E2 -6313.176} C_VEL
LIN {X 0,Y 497.486,Z 500.644,A -85,B 0,C 180,E1 -6313.74,E2 -6313.74} C_VEL
LIN {X 0,Y 497.716,Z 487.937,A -85,B 0,C 180,E1 -6314.15,E2 -6314.15} C_VEL
LIN {X 0,Y 497.855,Z 475.195,A -85,B 0,C 180,E1 -6314.407,E2 -6314.407} C_VEL
LIN {X 0,Y 498.482,Z 385.776,A -85,B 0,C 180,E1 -6315.793,E2 -6315.793} C_VEL
LIN {X 0,Y 496.528,Z 374.646,A -85,B 0,C 180,E1 -6316.045,E2 -6316.045} C_VEL
LIN {X 0,Y 496.915,Z 357.327,A -85,B 0,C 180,E1 -6318.984,E2 -6318.984} C_VEL
LIN {X 0,Y 497.202,Z 340.908,A -85,B 0,C 180,E1 -6321.78,E2 -6321.78} C_VEL
LIN {X 0,Y 495.779,Z 332.355,A -85,B 0,C 180,E1 -6323.319,E2 -6323.319} C_VEL
LIN {X 0,Y 495.829,Z 332.347,A -85,B 0,C 180,E1 -6326.749,E2 -6326.749} C_VEL
LIN {X 0,Y 495.771,Z 332.354,A -85,B 0,C 180,E1 -6329.746,E2 -6329.746} C_VEL
LIN {X 0,Y 495.773,Z 332.352,A -85,B 0,C 180,E1 -6332.594,E2 -6332.594} C_VEL
LIN {X 0,Y 495.75,Z 332.356,A -85,B 0,C 180,E1 -6335.538,E2 -6335.538} C_VEL
LIN {X 0,Y 495.763,Z 332.351,A -85,B 0,C 180,E1 -6338.767,E2 -6338.767} C_VEL
LIN {X 0,Y 495.743,Z 332.36,A -85,B 0,C 180,E1 -6341.897,E2 -6341.897} C_VEL
LIN {X 0,Y 495.742,Z 332.356,A -85,B 0,C 180,E1 -6345.14,E2 -6345.14} C_VEL
LIN {X 0,Y 495.725,Z 332.358,A -85,B 0,C 180,E1 -6345.435,E2 -6345.435} C_VEL
LIN {X 0,Y 495.047,Z 332.445,A -85,B 0,C 180,E1 -6346.112,E2 -6346.112} C_VEL
LIN {X 0,Y 492.185,Z 332.801,A -85,B 0,C 180,E1 -6347.213,E2 -6347.213} C_VEL
LIN {X 0,Y 489.776,Z 333.1,A -85,B 0,C 180,E1 -6348.1,E2 -6348.1} C_VEL
LIN {X 0,Y 488.748,Z 333.226,A -85,B 0,C 180,E1 -6348.785,E2 -6348.785} C_VEL
LIN {X 0,Y 488.667,Z 333.236,A -85,B 0,C 180,E1 -6349.017,E2 -6349.017} C_VEL
LIN {X 0,Y 488.663,Z 333.242,A -85,B 0,C 180,E1 -6351.797,E2 -6351.797} C_VEL
LIN {X 0,Y 488.72,Z 333.233,A -85,B 0,C 180,E1 -6355.053,E2 -6355.053} C_VEL
LIN {X 0,Y 488.687,Z 333.236,A -85,B 0,C 180,E1 -6358.049,E2 -6358.049} C_VEL
LIN {X 0,Y 488.693,Z 333.237,A -85,B 0,C 180,E1 -6360.727,E2 -6360.727} C_VEL
LIN {X 0,Y 488.67,Z 333.238,A -85,B 0,C 180,E1 -6363.522,E2 -6363.522} C_VEL
LIN {X 0,Y 488.701,Z 333.347,A -85,B 0,C 180,E1 -6365.078,E2 -6365.078} C_VEL
LIN {X 0,Y 491.016,Z 345.005,A -85,B 0,C 180,E1 -6367.265,E2 -6367.265} C_VEL
LIN {X 0,Y 490.477,Z 358.992,A -85,B 0,C 180,E1 -6369.666,E2 -6369.666} C_VEL
LIN {X 0,Y 490.281,Z 362.927,A -85,B 0,C 180,E1 -6370.332,E2 -6370.332} C_VEL
LIN {X 0,Y 493.575,Z 379.686,A -85,B 0,C 180,E1 -6370.727,E2 -6370.727} C_VEL
LIN {X 0,Y 492.551,Z 499.568,A -85,B 0,C 180,E1 -6372.509,E2 -6372.509} C_VEL
LIN {X 0,Y 492.225,Z 514.449,A -85,B 0,C 180,E1 -6372.902,E2 -6372.902} C_VEL
LIN {X 0,Y 491.844,Z 528.394,A -85,B 0,C 180,E1 -6373.447,E2 -6373.447} C_VEL
LIN {X 0,Y 491.349,Z 541.398,A -85,B 0,C 180,E1 -6374.123,E2 -6374.123} C_VEL
LIN {X 0,Y 490.774,Z 553.991,A -85,B 0,C 180,E1 -6374.955,E2 -6374.955} C_VEL
LIN {X 0,Y 490.208,Z 565.468,A -85,B 0,C 180,E1 -6375.892,E2 -6375.892} C_VEL
LIN {X 0,Y 489.667,Z 576.189,A -85,B 0,C 180,E1 -6376.955,E2 -6376.955} C_VEL
LIN {X 0,Y 489.27,Z 586.663,A -85,B 0,C 180,E1 -6378.216,E2 -6378.216} C_VEL
LIN {X 0,Y 488.73,Z 596.352,A -85,B 0,C 180,E1 -6379.644,E2 -6379.644} C_VEL
LIN {X 0,Y 488.412,Z 604.336,A -85,B 0,C 180,E1 -6381.1,E2 -6381.1} C_VEL
LIN {X 0,Y 488.178,Z 610.767,A -85,B 0,C 180,E1 -6382.554,E2 -6382.554} C_VEL
LIN {X 0,Y 488.064,Z 616.467,A -85,B 0,C 180,E1 -6384.214,E2 -6384.214} C_VEL
LIN {X 0,Y 487.943,Z 620.609,A -85,B 0,C 180,E1 -6385.869,E2 -6385.869} C_VEL
LIN {X 0,Y 487.907,Z 623.326,A -85,B 0,C 180,E1 -6387.522,E2 -6387.522} C_VEL
LIN {X 0,Y 487.831,Z 624.693,A -85,B 0,C 180,E1 -6389.173,E2 -6389.173} C_VEL
LIN {X 0,Y 487.831,Z 624.736,A -85,B 0,C 180,E1 -6390.824,E2 -6390.824} C_VEL
LIN {X 0,Y 487.906,Z 623.453,A -85,B 0,C 180,E1 -6392.475,E2 -6392.475} C_VEL
LIN {X 0,Y 487.942,Z 620.813,A -85,B 0,C 180,E1 -6394.129,E2 -6394.129} C_VEL
LIN {X 0,Y 488.061,Z 616.743,A -85,B 0,C 180,E1 -6395.784,E2 -6395.784} C_VEL
LIN {X 0,Y 488.174,Z 611.123,A -85,B 0,C 180,E1 -6397.443,E2 -6397.443} C_VEL
LIN {X 0,Y 488.402,Z 604.783,A -85,B 0,C 180,E1 -6398.897,E2 -6398.897} C_VEL
LIN {X 0,Y 488.698,Z 596.895,A -85,B 0,C 180,E1 -6400.355,E2 -6400.355} C_VEL
LIN {X 0,Y 489.127,Z 588.644,A -85,B 0,C 180,E1 -6401.603,E2 -6401.603} C_VEL
LIN {X 0,Y 489.607,Z 578.081,A -85,B 0,C 180,E1 -6402.928,E2 -6402.928} C_VEL
LIN {X 0,Y 490.125,Z 567.639,A -85,B 0,C 180,E1 -6404.002,E2 -6404.002} C_VEL
LIN {X 0,Y 490.652,Z 556.629,A -85,B 0,C 180,E1 -6404.94,E2 -6404.94} C_VEL
LIN {X 0,Y 491.19,Z 544.68,A -85,B 0,C 180,E1 -6405.773,E2 -6405.773} C_VEL
LIN {X 0,Y 491.749,Z 531.473,A -85,B 0,C 180,E1 -6406.501,E2 -6406.501} C_VEL
LIN {X 0,Y 492.159,Z 517.827,A -85,B 0,C 180,E1 -6407.072,E2 -6407.072} C_VEL
LIN {X 0,Y 492.496,Z 503.555,A -85,B 0,C 180,E1 -6407.49,E2 -6407.49} C_VEL
LIN {X 0,Y 492.746,Z 483.76,A -85,B 0,C 180,E1 -6407.829,E2 -6407.829} C_VEL
LIN {X 0,Y 493.549,Z 379.091,A -85,B 0,C 180,E1 -6409.374,E2 -6409.374} C_VEL
LIN {X 0,Y 490.299,Z 362.826,A -85,B 0,C 180,E1 -6409.775,E2 -6409.775} C_VEL
LIN {X 0,Y 491.036,Z 346.812,A -85,B 0,C 180,E1 -6412.509,E2 -6412.509} C_VEL
LIN {X 0,Y 490.771,Z 343.4,A -85,B 0,C 180,E1 -6413.12,E2 -6413.12} C_VEL
LIN {X 0,Y 488.674,Z 333.242,A -85,B 0,C 180,E1 -6415.034,E2 -6415.034} C_VEL
LIN {X 0,Y 488.677,Z 333.241,A -85,B 0,C 180,E1 -6417.399,E2 -6417.399} C_VEL
LIN {X 0,Y 488.685,Z 333.238,A -85,B 0,C 180,E1 -6420.357,E2 -6420.357} C_VEL
LIN {X 0,Y 488.722,Z 333.233,A -85,B 0,C 180,E1 -6423.482,E2 -6423.482} C_VEL
LIN {X 0,Y 488.665,Z 333.239,A -85,B 0,C 180,E1 -6426.351,E2 -6426.351} C_VEL
LIN {X 0,Y 488.679,Z 333.238,A -85,B 0,C 180,E1 -6429.254,E2 -6429.254} C_VEL
LIN {X 0,Y 488.658,Z 333.237,A -85,B 0,C 180,E1 -6431.593,E2 -6431.593} C_VEL
LIN {X 0,Y 488.691,Z 333.238,A -85,B 0,C 180,E1 -6434.801,E2 -6434.801} C_VEL
LIN {X 0,Y 488.656,Z 333.238,A -85,B 0,C 180,E1 -6437.47,E2 -6437.47} C_VEL
LIN {X 0,Y 488.683,Z 333.239,A -85,B 0,C 180,E1 -6440.744,E2 -6440.744} C_VEL
LIN {X 0,Y 488.656,Z 333.236,A -85,B 0,C 180,E1 -6443.866,E2 -6443.866} C_VEL
LIN {X 0,Y 488.689,Z 333.232,A -85,B 0,C 180,E1 -6446.873,E2 -6446.873} C_VEL
